FUNCTION FC 8 : VOID
TITLE = Ermittlung DB, DW, Laenge Anyzeiger
//Erstellung:
//Datum        Bearbeiter                                                 Version
//--------------------------------------------------------------------------------
//03.03.99     A.Geiger (gea)                                             01.00.00
//
//Änderungen:
//Nr. Datum    Bearb Beschreibung                                   Marke Version
//--------------------------------------------------------------------------------
//01  
//
//________________________________________________________________________________
//Funktion:
//
//Der Baustein ermittelt aus einem ANY-Zeiger:
//  Datenbausteinnummer
//  Datenwortnummer Beginn des Anyzeigers
//  Länge des Bereiches in Byte
//
AUTHOR : gea
FAMILY : AZO
VERSION : 0.0
VAR_INPUT
  in_Zeiger : ANY ;	//ANY-Zeiger
END_VAR
VAR_OUTPUT
  out_DB : INT ;	//Datenbausteinnummer
  out_DW : INT ;	//Anfangs-Datenwortnummer
  out_Laenge : INT ;	//Länge des Bereiches in Byte
END_VAR
BEGIN
NETWORK
TITLE = Ermittlung DB, DW, Laenge Anyzeiger
      L     P##in_Zeiger;
      LAR1;
      L     W [AR1,P#2.0];
      T     #out_Laenge;
      L     W [AR1,P#4.0];
      T     #out_DB;
      L     D [AR1,P#6.0];
      SRD   3;
      T     #out_DW;
END_FUNCTION

FUNCTION FC 10 : VOID
TITLE = Analogwert lesen/schreiben
//Erstellung:
//Datum        Bearbeiter                                                 Version
//--------------------------------------------------------------------------------
//06.08.97     G.Herkert (hkt)                                            01.00.00
//
//Änderungen:
//Nr. Datum    Bearb Beschreibung                                   Marke Version
//--------------------------------------------------------------------------------
//01  21.10.97 rh    Drahtbruchüberwachung ergänzt                        01.01.00
//02  05.12.97 rh    Adressen auf PEW und PAW geändert                    01.01.01
//03  25.11.98 gea   Simulation eingefügt                                 01.02.00
//04  29.03.99 gea   Fehlerbehebung Drahtbruchüberwachung                 01.02.01
//05  30.06.99 sra   Fehlerbehebung Drahtbruchüberwachung                 01.02.02
//06  19.02.00 sra   Unterscheidung Drahtbruchüberwachung                 01.02.03
//07  12.09.01 gea   Eingangsparameter in_E_A_Adresse als INT             01.03.00
//08  16.03.04 sra   nicht in Simulations-DB schreiben wenn Simul aus     01.03.01
//09  17.09.08 sra   Wago-System 750-466 erweitert                  (009) 01.04.00
//________________________________________________________________________________
//Funktion:
//
//Der Baustein liest den Wert eines Analogeinganges ein und normiert diesen. Die 
//Normierung erfolgt anhand der Vorgabe der Eingangsparameter Obergrenze und 
//Untergrenze.
//
//Hinweis:
//- bei Siemens-Baugruppen ist der Wert "MaxDigit" = 27648
//- bei Wago-Baugruppen 740-466 ist der Wert "MaxDigit" = 32760
//
//
AUTHOR : hkt
FAMILY : AZO
VERSION : 0.0
VAR_INPUT
  in_E_A : CHAR  := 'E';	//E = Eingang, A = Ausgang
  in_EA_Adresse : INT ;	//Ein-/Ausgangsadresse des Analogkanals
  in_OberGrenze : REAL ;	//Obergrenze des Ausgabewertes (z.B. Drucktransmitter: 2 bar)
  in_UnterGrenze : REAL ;	//Untergrenze des Ausgabewertes (z.B. Drucktransmitter: 0 bar)
  in_MaxDigit : REAL ;	//Digitwert den die Baugruppe bei der Obergrenze liefert z.B. 27648
  in_MinDigit : REAL ;	//Digitwert den die Baugruppe bei der Untergrenze liefert z.B. 0 bzw. -27648
  in_Typ : CHAR ;	//Z=Zentralbaugruppe, B=ET200B Analogmodul, W=Wago 750-466, sonstige
  in_Simulation : BOOL ;	//Simulation des Analogwertes über Eintrag in Datenbaustein
  in_DB_Simulation_EA : INT ;	//Simulation-DB des Analogwertes über Eintrag in Datenbaustein
END_VAR
VAR_IN_OUT
  io_Wert : REAL ;	//eingelesener und normierter Wert den die Baugrppe liefert
  io_Drahtbruch : BOOL ;	//Drahtbruchstoerung
END_VAR
VAR_TEMP
  MaxDigit_MinDigit : REAL ;
  E_MinDigit : REAL ;
  OG_UG : REAL ;
  Eingang_Real : REAL ;
  Pointer_EA_Adresse : DWORD ;
  Wert_analog : WORD ;
  DB_Sim : INT ;
END_VAR
BEGIN
NETWORK
TITLE = Zwischenwerte berechnen
      L     #in_MaxDigit;
      L     #in_MinDigit;
      -R;
      T     #MaxDigit_MinDigit;
      L     #in_OberGrenze;
      L     #in_UnterGrenze;
      -R;
      T     #OG_UG;
NETWORK
TITLE = Zeiger berechnen
// Zeiger auf EA-Adresse berechnen
      LAR1  P#0.0;
      L     #in_EA_Adresse;
      SLW   3;
      +AR1;
      LAR1;
      T     #Pointer_EA_Adresse;	//Zeiger auf EA-Adresse
      L     #in_DB_Simulation_EA;
      T     #DB_Sim;	//Zeiger auf EA-DB
NETWORK
TITLE = Analogwert einlesen
//Analogwert einlesen
//Formel:   Wert = UG + (OG-UG)*(E-MinDigit) / (MaxDigit-MminDigit)
      L     #in_E_A;
      L     'E';
      <>I;
      JC    NotE;
      A     #in_Simulation;
      JC    SIME;
      L     PIW [#Pointer_EA_Adresse];
      JU    WERE;	// (008)
SIME: OPN   DB [#DB_Sim];
      L     DBW [#Pointer_EA_Adresse];
WERE: T     #Wert_analog;
      A(;
      L     #in_Typ;	// Abfrage Drahtbruchüberwachung
      L     'Z';	// "Z" = Zentralbaugruppe
      ==I;
      );
      A(;
      L     #Wert_analog;	// 7FFF Ersatzwert für Drahtbruch
      L     W#16#7FFF;
      ==I;
      );
      O;
      A(;
      L     #in_Typ;	// Abfrage Drahtbruchüberwachung
      L     'B';	// "B" = ET200B Baugruppe
      ==I;
      );
      A(;
      L     #Wert_analog;	// 8000 Ersatzwert für Drahtbruch
      L     W#16#8000;
      ==I;
      );
      O;	// -> (009)
      A(;
      L     #in_Typ;	// Abfrage Kartentyp
      L     'W';	// "W" = Wago System 750-466
      ==I;	// Karte meldet mit den rechten 3 Bis ein Kurzschluss bzw. Überlauf
      );
      A(;
      L     #Wert_analog;
      L     W#16#7;
      AW;
      L     W#16#0;
      <>I;
      );	// <- (009)
      =     #io_Drahtbruch;
      L     #Wert_analog;
      ITD;
      DTR;
      T     #Eingang_Real;
      L     #Eingang_Real;
      L     #in_MinDigit;
      -R;
      T     #E_MinDigit;
      L     #OG_UG;
      L     #E_MinDigit;
      *R;
      L     #MaxDigit_MinDigit;
      /R;
      L     #in_UnterGrenze;
      +R;
      T     #io_Wert;
NotE: NOP   0;
NETWORK
TITLE = AnalogWert ausgeben:  
//AnalogWert ausgeben:
//Formel : A = MinDigit+(MaxDigit-MinDigit)*(Wert-UG)/ (Og-UG)
      L     #in_E_A;
      L     'A';
      <>I;
      JC    NotA;
      L     #io_Wert;
      L     #in_UnterGrenze;
      -R;
      L     #OG_UG;
      /R;
      L     #MaxDigit_MinDigit;
      *R;
      L     #in_MinDigit;
      +R;
      RND;
      T     #Wert_analog;
      A     #in_Simulation;
      JC    SIMA;
      T     PQW [#Pointer_EA_Adresse];
      JU    NotA;	// (008)
SIMA: OPN   DB [#DB_Sim];
      T     DBW [#Pointer_EA_Adresse];
NotA: NOP   0;
END_FUNCTION

FUNCTION FC 13 : VOID
TITLE = Baustein für Standardmerker
//Erstellung:
//Datum        Bearbeiter                                                 Version
//--------------------------------------------------------------------------------
//26.06.97     R.Schaffert (sra)                                          01.00.00
//
//Änderungen:
//Nr. Datum    Bearb Änderung                                       Marke  Version
//--------------------------------------------------------------------------------
//01  21.11.02 sra   Resetmerker eingefügt                          (001) 01.00.01
//02  30.08.12 pti   Lampe Steuerspannung ein eingefügt             (002) 01.01.00
//03  23.07.13 sra   Signale für Sicherung eingefügt                (003) 01.02.00
//04  05.12.13 sra   Signal Steuerspannung gelöscht                       01.03.00
//05  02.06.14 sra   M0.3 Reset ebenfalls gelöscht (zu Änderung 04)       01.03.01
//06  14.12.16 sra   Implement SFC51 to read battery information    (006) 01.04.00
//________________________________________________________________________________
//Funktion:
//  
//Der Baustein erzeugt folgende Standardsignale:
//- M 0.1 "konstant 1" Merker
//- M 0.2 "konstant 0" Merker
//- M 1.6 Melderentprelltakt (5 Sekunden) 
//- M 1.7 "Takt Timernachbildung" = in_Basistakt_Timer
//- MB4 Impulsmerker für Takte 2.0s, 1.6s, 1.0s, 0.8s, 0.5s, 0.4s, 0.2s, 0.1s
//  !!! MB 2 muss als Taktmerker in CPU parametriert werden  !!
//  Das MB 3 wird als Hilfsbyte zur Flankenauswertung benutzt
//- MW 6 Zeitwert Takt = in_Zeit_Basistakt_100ms
AUTHOR : sra
FAMILY : AZO
VERSION : 0.0
VAR_INPUT
  in_E_Sicherung_OK : BOOL ;	//Eingang Sicherung OK = Eingang Störung Sicherung
  in_Basistakt_Timer : BOOL ;	//Taktmerker für alle Zeitfunktionen (abhängig von Zykluszeit)
  in_Zeit_Basistakt_100ms : INT ;	//Zeitwert Basistakt in 100 ms
END_VAR
VAR_OUTPUT
  o_Lampe_Stoer_Sicherung : BOOL ;	//Ausgang der Lampe "Störung Sicherung"
  o_Stoerung_Sicherung : BOOL ;	//Störung Sicherung -> für Störbitzuweisung im DB34
END_VAR
VAR_TEMP
  NOP : INT ;
END_VAR
BEGIN
NETWORK
TITLE = Statische Merker  
      SET;
      S     M 0.1;
      R     M 0.2;
NETWORK
TITLE = Lampe "Störung Sicherung" und Störmeldung Sicherung
//(003)
      AN    #in_E_Sicherung_OK;
      =     #o_Lampe_Stoer_Sicherung;
      =     #o_Stoerung_Sicherung;
NETWORK
TITLE = Impulsmerker Takte
//Impulsmerker für Takte 2.0s, 1.6s, 1.0s, 0.8s, 0.5s, 0.4s, 0.2s, 0.1s
//positive Flankenauswertung auf die von der CPU erzeugten Takte
      L     MB 3;
      L     MB 2;
      T     MB 3;
      XOW;
      L     MB 2;
      AW;
      T     MB 4;
NETWORK
TITLE = Werte für Timernachbildung vorgeben
//!! Abhängig von Zykluszeit !! 
      A     #in_Basistakt_Timer;
      =     M 1.7;
      L     #in_Zeit_Basistakt_100ms;
      T     MW 6;
NETWORK
TITLE = Takt Melderentprellung
//Takt Melderentprellung
      AN    M 1.6;
      L     S5T#5S;
      SD    T 1;
      A     T 1;
      =     M 1.6;
NETWORK
TITLE = read Battery fault of CPU
//(006)
      CALL  SFC 51 (
           REQ                      := M 2.7,
           SZL_ID                   := W#16#392,
           INDEX                    := W#16#0,
           RET_VAL                  := DB3.DBW 62,
           BUSY                     := DB3.DBX 60.0,
           SZL_HEADER               := P#DB3.DBX 64.0,
           DR                       := P#DB3.DBX 68.0 BYTE 20);	// W#16#392 = Status of the backup batteries in a rack/module rack of a CPU after at least one battery has failed /  if ID = 392h -> Index is always 0
      L     DB3.DBB 68;
      L     0;
      <>I;
      =     DB3.DBX 31.3;
END_FUNCTION

FUNCTION FC 16 : VOID
TITLE = Sammelstoerung
//Erstellung:
//Datum        Bearbeiter                                                 Version
//--------------------------------------------------------------------------------
//26.07.99     M.Junker (jm)                                              01.00.00
//
//Änderungen:
//Nr. Datum    Bearb Änderung                                       Marke  Version
//--------------------------------------------------------------------------------
//01  14.09.99 jm    Spiegelung von PC ergänzt                            01.01.00
//02  06.10.99 jm    Störauswertung DWORD-weise                           01.02.00
//03  23.10.99 jm    QuitierungsDWORD von PC löschen                      01.03.00
//04  03.11.99 jm    Fehlerbeseitigung: QIP und DWORD                     01.03.01
//05  27.03.00 jm    Fehlerbeseitigung DWORD (Erstmeldung)                01.03.02
//06  19.04.05 jm    Fehlerbeseitigung Pointeradressen >8192(=>SLD) (006) 01.03.03
//07  23.02.06 jm    Quittierungs-DB Farbgrafik ist extern
//                   => Quittierung üder Kastor oder Farbgrafik     (007) 01.04.00
//08  23.03.06 sra   Einzelstörungsbereiche
//                   +Quitt.Erstwertmeldung über Quittierbereich         
//                   +Erstwertmeldung löschen ohne Störung          (008) 01.05.00
//09  10.05.06 sra   Fehlerbeseitigung zu Änderung 08               (009) 01.05.01
//10  11.05.06 sra   Änderung Quittierung von Farbgrafik            (010) 01.05.02
//11  05.10.06 jm    Anpassung für Siemens OP: extra Quittierbereich
//                   mit Flankenauswertung                          (011) 01.06.00
//12  01.04.08 jm    Steuerspannung entfernt, da Probleme mit OP-
//                   Quittierung (Problem: vorhandene Störung bei
//                   Steuerspannung aus am OP quittieren)           (012) 01.06.01
//13  16.11.15 sra   "Steuerspannung" in "Frg. Sammenstörung" geänd.(013) 01.06.02
//________________________________________________________________________________
//Beschreibung:
//
//!!!ACHTUNG: Parameter Anzahl Störungsbyte muß immer durch 4 teilbar sein!!!!
//
//Der Baustein überwacht einen definierbaren Teil eines Datenbaustein (DB34) in 
//dem alle Störmeldungen gesammelt werden. Sobald eine Störung vorhanden ist wird 
//das Signal "Sammelstörung" gebildet um damit z.B. eine Sammelstörlampe 
//anzusteuern. Der Parameter "Anzahl Störungsbyte" muß immer durch 4 teilbar sein
//
//In weiteren Bereichen weden die Datenblöcke "Erstmeldung", "Erstmeldung PC" und 
//Quittierung PC" mit der gleichen Größe wie der Störbereich benötigt.
//
//Funktion:
//Um bei der Störungsquittierung zur FG kompatibel zu sein werden die 
//Quittierungen, sobald die Störung verschwunden ist, von der SPS gelöscht.
//
//Die beiden Quittierungsbereiche (in DB34 für Kastor; in DB35 für SCADA) werden 
//mit ODER ausgewertet, d.h. die Störungen könnten von beiden Seiten quittiert 
//werden (wird normal nicht gemacht). Die Quittierbits werden hier so umkopiert, 
//daß sie immer in beiden Quittierungsbereichen auftauchen.
//=> es müssen immer beide Quittierbereiche angelegt sein
//=> an den Aggregat-Baustein werden die Bits aus dem DB35 angelegt
//
//OP:
//Siemens OPs müssen in einen extra Bereich quittieren, der hinter dem normalen 
//Standardbereichen im DB34 liegt. Im Anschluss folgt noch ein Bereich für die 
//Flankenauswertung. Bei positiver Flanke der Quittierung von OP wird die in den 
//Bereich der SCADA-Quittierung übertragen. In den OP Quittierbereich darf auf 
//gar keinen Fall die SPS schreiben. Wird kein OP verwendet so können die 
//OP-Bereiche aus dem DB34 weggelassen werden.
AUTHOR : jm
FAMILY : STANDARD
NAME : hsh
VERSION : 0.0
VAR_INPUT
  Conf_AckBySiemensOP : BOOL ;	//configuration bit: ackowledge done by Siemens OP (011)
  Stoerungstakt : BOOL ;	//Takt für Störauswertung
  Freigabe_Sammelstoerung : BOOL ;	//Freigabe Sammelstörung (ehemals Steuerspannung)
  Quittierung : BOOL ;	//Quittierung Fehlermeldung
  Stoerungs_DB : INT ;	//Stör-Datenbaustein
  Quittierungs_DB_SCADA : INT ;	//Quittier-Datenbaustein Farbgrafik
  Anzahl_Stoerungs_Byte : INT ;	//Anzahl Störungsbyte im Stör-Db (Blocklänge der 4 Bereiche)
  Offset_Stoerungs_Byte : INT ;	//Anfangs-DW der Störmeldungen im Stör-DB (wenn Bereich nicht bei Byte 0 anfängt)
  Adresse_Anfangswort : INT ;	//Adresse des ersten Datenwortes das ausgewertet wird
  Bereichslaenge : INT ;	//Länge des Bereiches der ausgewertet wird (!!Muss durch 4 teilbar sein!!)
END_VAR
VAR_IN_OUT
  Sammelstoerung : BOOL ;	//Sammelstörung
  Erstmeldung : BOOL ;	//Erstmeldung aktiv
  Erstmeldung_PC : BOOL ;	//Erstmeldung an PC
  Quittierung_PC : BOOL ;	//Quittierung von PC
END_VAR
VAR_TEMP
  Stoer_DB : INT ;	//Stoerungs-DB lokal
  Quit_DB : INT ;	//Quittierungs-DB extern
  Offsetende : INT ;	//= Störungsbyte + Offset
  SI : INT ;	//Störungsindex
  KI : INT ;	//Kopierindex
  SIP : INT ;	//Spiegelungsindex PC
  QIP : INT ;	//Quittierungsindex PC
  QIS : INT ;	//Quitierungsindex SCADA
  QIO : INT ;	//Quittierungsindex Siemens OP (011)
  KQIO : INT ;	//Kopie Quittierungsindex Siemens OP (011)
  StoerungsDWORD : DWORD ;	//Stoerungsdoppelwort
  KopieDWORD : DWORD ;	//Kopiedoppelwort
  SpiegelungsDWORD : DWORD ;	//Spiegelungsdoppelwort
  QuittierungsDWORD : DWORD ;	//Quittierungsdoppelwort
  QuitPC_DWORD : DWORD ;	//Quittierungsdoppelwort von PC
  QuitSCADA_DWORD : DWORD ;	//Quittierungsdoppelwort von SCADA
  QuitOP_DWORD : DWORD ;	//Quittierungdoppelwort von OP (011)
  KopieQuitOP_DWORD : DWORD ;	//Kopie Quittierungdoppelwort von OP (011)
  t_Erstmeldung_PC : BOOL ;	//Erstmeldung an PC
END_VAR
BEGIN
NETWORK
TITLE = Störauswertung aktiv?
//      ON    #Steuerspannung // (012)
//      SPB   FCEN                       // FunCtion ENd // (012)
      ON    #Stoerungstakt;
      JC    QUIT;	// QUITtierung Erstmeldung prüfen
NETWORK
TITLE = Variablen vorbelegen
//Minus 4 wegen DWORD-Auswertung
      CLR;
      =     #Sammelstoerung;
      =     #t_Erstmeldung_PC;
      L     #Offset_Stoerungs_Byte;
      L     #Adresse_Anfangswort;	// (008)
      +I;	// (008)
      L     #Bereichslaenge;	// (008)
      +I;
      T     #Offsetende;	//Offsetende = Offset + Anzahl // (007)
      L     #Offsetende;	// (007)
      L     4;
      -I;
      T     #SI;	//Stoerungsindex = Offsetende + Anzahl -4
      T     #QIS;	//Quittierungsindex SCADA = Stoerungsindex (007)
      L     #Offsetende;	// (007)
      L     #Anzahl_Stoerungs_Byte;	// (008)
      +I;
      L     4;
      -I;
      T     #KI;	//Kopierindex = Offsetende + Anzahl*2 -4
      L     #Offsetende;	// (007)
      L     #Anzahl_Stoerungs_Byte;
      +I;
      L     #Anzahl_Stoerungs_Byte;	// (008)
      +I;
      L     4;
      -I;
      T     #SIP;	//Spiegelungsindex PC = Offsetende + Anzahl*3 -4
      L     #Offsetende;	// (007)
      L     #Anzahl_Stoerungs_Byte;
      +I;
      L     #Anzahl_Stoerungs_Byte;
      +I;
      L     #Anzahl_Stoerungs_Byte;	// (008)
      +I;
      L     4;
      -I;
      T     #QIP;	//Quittierungsindex PC = Offsetende + Anzahl*4 -4
// >>>>>>>>>> (011)
      L     #Offsetende;
      L     #Anzahl_Stoerungs_Byte;
      +I;
      L     #Anzahl_Stoerungs_Byte;
      +I;
      L     #Anzahl_Stoerungs_Byte;
      +I;
      L     #Anzahl_Stoerungs_Byte;
      +I;
      L     4;
      -I;
      T     #QIO;	//Quittierungsindex OP = Offsetende + Anzahl*5 -4
      L     #Offsetende;
      L     #Anzahl_Stoerungs_Byte;
      +I;
      L     #Anzahl_Stoerungs_Byte;
      +I;
      L     #Anzahl_Stoerungs_Byte;
      +I;
      L     #Anzahl_Stoerungs_Byte;
      +I;
      L     #Anzahl_Stoerungs_Byte;
      +I;
      L     4;
      -I;
      T     #KQIO;	//Kopie Quittierungsindex OP = Offsetende + Anzahl*6 -4
// <<<<<<<<<< (011)
NETWORK
TITLE = Störungs-/Kopie-/Spiegelungs-/QuittierungsDWORD(OP) laden
      L     #Stoerungs_DB;
      T     #Stoer_DB;
      L     #Quittierungs_DB_SCADA;	// (007)
      T     #Quit_DB;	// (007)
SLOP: OPN   DB [#Stoer_DB];
      L     #SI;
      SLD   3;	// (006)
      LAR1;
      L     DBD [AR1,P#0.0];
      T     #StoerungsDWORD;
      L     #KI;
      SLD   3;	// (006)
      LAR1;
      L     DBD [AR1,P#0.0];
      T     #KopieDWORD;
      L     #SIP;
      SLD   3;	// (006)
      LAR1;
      L     DBD [AR1,P#0.0];
      T     #SpiegelungsDWORD;
      L     #QIP;
      SLD   3;	// (006)
      LAR1;
      L     DBD [AR1,P#0.0];
      T     #QuitPC_DWORD;	// (007)
///*(007)
      L     L#0;	// (011)
      T     #QuitSCADA_DWORD;
      L     #Quittierungs_DB_SCADA;	// (011)
      L     0;
      ==I;	// (011)
      JC    KQ1;	// (011) kein Quittierungsbaustein vorhanden
      OPN   DB [#Quit_DB];
      L     #QIS;
      SLD   3;
      LAR1;
      L     DBD [AR1,P#0.0];
      T     #QuitSCADA_DWORD;
      OPN   DB [#Stoer_DB];
//(007)*/
// >>>>>>>>>> (011)
      L     0;
      T     #QuitOP_DWORD;	// vorbelegen, falls nicht vorhanden
      AN    #Conf_AckBySiemensOP;
      JC    NOPA;	// No OP Acknowledge
      L     #QIO;
      SLD   3;
      LAR1;
      L     DBD [AR1,P#0.0];
      T     #QuitOP_DWORD;
      L     #KQIO;
      SLD   3;
      LAR1;
      L     DBD [AR1,P#0.0];
      T     #KopieQuitOP_DWORD;
NOPA: NOP   0;	// No OP Acknowledge
// <<<<<<<<<< (011)
KQ1:  NOP   0;
NETWORK
TITLE = Pos.Flanke Quittierung OP
//(011)
      AN    #Conf_AckBySiemensOP;
      JC    NPOA;	// No Processing of Op Acknowledge
      L     #QuitOP_DWORD;	// -
      L     #KopieQuitOP_DWORD;	// |
      XOD;	// | positive Flanke Quittierung OP
      L     #QuitOP_DWORD;	// |
      AD;	// -
      L     #QuitSCADA_DWORD;
      OD;
      T     #QuitSCADA_DWORD;	// => Quittierung in QuitSCADA setzen
      L     #QuitOP_DWORD;
      T     #KopieQuitOP_DWORD;	// => Hilfsmerker Flanke (Kopie ALT)
NETWORK
TITLE = Quittierung OP DWORD nach Kopiebyte
//(011)
      L     #KQIO;
      SLD   3;
      LAR1;
      L     #KopieQuitOP_DWORD;
      T     DBD [AR1,P#0.0];	// => Quittierung OP merken
NPOA: NOP   0;
NETWORK
TITLE = Sammelstörung
      L     #StoerungsDWORD;
      L     0;
      <>D;
      A     #Freigabe_Sammelstoerung;	// (012)
      S     #Sammelstoerung;
NETWORK
TITLE = Erstwertmeldung
      L     #StoerungsDWORD;
      L     #KopieDWORD;
      XOD;
      L     #StoerungsDWORD;
      AD;
      L     0;
      <>D;
      A     #Freigabe_Sammelstoerung;	// (012)
      S     #Erstmeldung;
NETWORK
TITLE = Erstwertmeldung an PC
      L     #StoerungsDWORD;
      L     #SpiegelungsDWORD;
      <>D;
      S     #t_Erstmeldung_PC;
NETWORK
TITLE = StoerungsDWORD nach Kopiebyte
      L     #KI;
      SLD   3;	// (006)
      LAR1;
      L     #StoerungsDWORD;
      T     DBD [AR1,P#0.0];
NETWORK
TITLE = neue Quittierung?
//(008)
      L     #QuitSCADA_DWORD;
      L     #QuitPC_DWORD;
      XOD;
      L     0;
      <>D;
      R     #Erstmeldung;
NETWORK
TITLE = QuittierungsDWORD bilden
//(007)
      L     #QuitPC_DWORD;	// (010)
      L     #SpiegelungsDWORD;	// (010)
      AD;	// (010)
      L     #QuitSCADA_DWORD;
      OD;
      T     #QuittierungsDWORD;	// Quittierung von Kastor oder SCADA
NETWORK
TITLE = QuittierungsDWORD löschen
      L     #StoerungsDWORD;
      L     #QuittierungsDWORD;
      AD;
      T     #QuittierungsDWORD;
NETWORK
TITLE = QuittierungsDWORD PC und SCADA löschen
      L     #QIP;
      SLD   3;	// (006)
      LAR1;
      L     #QuittierungsDWORD;
      T     DBD [AR1,P#0.0];	// PC Quittierung
      L     #Quittierungs_DB_SCADA;	// (011)
      L     0;	// (011)
      ==I;	// (011)
      JC    KQ2;	// (011) kein Quittierungsbaustein vorhanden
///*(007)
      OPN   DB [#Quit_DB];
      L     #QIS;
      SLD   3;
      LAR1;
      L     #QuittierungsDWORD;
      T     DBD [AR1,P#0.0];	// SCADA Quittierung
//(007)*/
KQ2:  NOP   0;
NETWORK
TITLE = Störungsschleife von (Anzahl - 4) bis 0
//Minus 4 wegen DWORD-Auswertung
// >>>>>>>>>> (011)
      L     #KQIO;
      L     4;
      -I;
      T     #KQIO;
      L     #QIO;
      L     4;
      -I;
      T     #QIO;
// <<<<<<<<<< (011)
///*(007)
      L     #QIS;
      L     4;
      -I;
      T     #QIS;
//(007)*/
      L     #QIP;
      L     4;
      -I;
      T     #QIP;
      L     #SIP;
      L     4;
      -I;
      T     #SIP;
      L     #KI;
      L     4;
      -I;
      T     #KI;
      L     #SI;
      L     4;
      -I;
      T     #SI;
      L     #Offset_Stoerungs_Byte;
      L     #Adresse_Anfangswort;	// (008)
      +I;	// (008)
      L     #SI;	// (008)
      <=I;	// (008) (009)
      JC    SLOP;	// Störungs LOOP
NETWORK
TITLE = Störauswertung für PC aktiv?
      O     #Erstmeldung_PC;
      O     #Quittierung_PC;
      JC    QUIT;	//QUITtierung
      A     #t_Erstmeldung_PC;
      S     #Erstmeldung_PC;
NETWORK
TITLE = Erstmeldung quittiert?
QUIT: A     #Quittierung;	//QUITtierung
      ON    #Sammelstoerung;	// (008)
      R     #Erstmeldung;
      A     #Quittierung_PC;
      R     #Erstmeldung_PC;
      NOP   0;
END_FUNCTION

FUNCTION FC 20 : VOID
TITLE = Block for motor actuation and fault monitoring
//Erstellung:
//Datum        Bearbeiter                                                 Version
//--------------------------------------------------------------------------------
//26.06.97     H.Rüttling (rh)                                            01.00.00
//
//Änderungen:
//Nr. Datum    Bearb Änderung                                       Marke  Version
//--------------------------------------------------------------------------------
//01  09.02.99 sra   Einfügen der Handbedienuung                    ()    01.01.00
//02  16.04.99 sra   Fehlerbeseitigung Störungsquittierung          ()    01.01.01
//03  23.07.99 sra   Ausg. wird auch bei Simulation gesetzt         ()    01.01.02
//04  19.10.99 sra   "in" Reparaturschalter gelöscht                ()    01.02.00
//05  03.11.99 hus   Parameter eingefügt "FU in Betrieb"            ()    01.03.00
//06  18.09.00 sra   komplette Überarbeitung / neue Struktur        ()    02.00.00
//07  08.11.02 sra   Änderung Betriebsstundenzähler (zählt falsch)  (007) 02.01.00
//08  31.10.05 sra   Ansteuerung Handbedienung im Automode rücksetz.
//                   Handbedienung zentral sperren                  (008) 02.02.00
//09  04.09.06 sra   Änderung Störungsquittierung                   (009) 02.03.00
//10  20.11.07 gea   Handmode zurücksetzen wenn Handmode gesperrt   (010) 02.03.01
//11  18.02.09 kmj   Objektststatus für OP ergänzt                  (011) 02.04.00
//12  20.03.09 kal   Objektststatus für OP ergänzt (überarbeitet)   (012) 02.04.01
//13  05.12.13 sra   "Anlage ein" eingefügt (Not-Aus-Konzept)       (013) 02.05.00
//________________________________________________________________________________
//Funktion:
//
//-Der Baustein steuert den Ablauf eines Motors mit 1 Ausgang und 1 Eingang durch 
// setzten des Eingangsparameters "in_Ansteuerung_Motor".
//
//-Der Ausgang wird nur angesteuert wenn der Eingang "in_Anlage_ein" = true
// ist. Diese Funktion ist vorhanden, um bei einem Not-Halt die Anlage vor 
// unkontrolliertem Einschalten zu schützen. 
//
//-Ist in der Motorstruktur die Taktfunktion freigegeben wird bei Freigabe des 
// Motors der Ausgang entsprechend der Impuls-/Pausezeit angesteuert.
// !!Der Baustein arbeitet nur mit vollen Sekunden!!
//
//-Der Baustein überwacht den Zustand des Ausgangs und des Eingangs und generiert 
// nach Ablauf der "Sollzeit Störung" eine Störmeldung
//
//-Ist das Bit "Simulation" auf TRUE, so wird der Eingang simuliert.
//
//-Ist die Kennung "Betriebsstundenzähler_ein" aktiviert werden die Laufzeit 
// des Motors aufsummiert. Dies erfolgt mit setzen des Ausgangs.
//
//-Der Baustein kopiert die Parameter "in_Eingang_Motor", "io_Ausgang_Motor", 
// "in_Quitt_Stoerung" und "io_Stoerung" in die angegebene Datenstruktur zur 
// Visualisierung auf einem Farbgrafiksystem. Diese Parameter müssen folglich 
// nicht mehr extern umkopiert werden.
//
//-Ist der Parameter "in_Handbedienung_erlaubt" angewählt kann der Motor über 
// eine Farbgrafik oder ein Bedienterminal manuell angesteuert werden
//
AUTHOR : rh
FAMILY : AZO
VERSION : 0.0
VAR_INPUT
  in_Handbedienung_erlaubt : BOOL ;	//1 = manual operation permitted, 0 = manual operation not permitted/locked
  in_Quitt_Stoerung_noetig : BOOL ;	//1 = fault acknowledgement required, 0 = automatic fault acknowledgement
  in_Anlage_ein : BOOL ;	//Anlage bzw. Anlagenbereich nach Not-Halt freigegeben
  in_Quitt_Stoerung : BOOL ;	//Fault acknowledgement when fault_acknowledgement_required = 1
  in_Ansteuerung_Motor : BOOL ;	//Actuation of motor in automatic mode
  in_Eingang_Motor : BOOL ;	//Input of motor
END_VAR
VAR_IN_OUT
  io_Ausgang_Motor : BOOL ;	//Output of motor
  io_Motor_in_Betrieb : BOOL ;	//Signal "motor in operation"
  io_Stoerung : BOOL ;	//Signal "motor fault"
  io_Motorstruktur : ANY ;	//ANY pointer of motor structure
END_VAR
VAR_TEMP
  Freigabe_Takt : BOOL ;
  Start_mit_Impuls : BOOL ;
  Dauertakt : BOOL ;
  Taktausgang : BOOL ;
  Taktanzahl_erreicht : BOOL ;
  Diskrepanz : BOOL ;
  Impulszeit : REAL ;
  Pausezeit : REAL ;
  Sollanzahl_Takte : INT ;
  Zeitzaehler : REAL ;
  Taktzaehler : INT ;
  Objektstatus : INT ;
END_VAR
BEGIN
NETWORK
TITLE = Anfangs-DW der Struktur aus ANY-Zeiger auslesen
      L     P##io_Motorstruktur;
      LAR2;
      L     D [AR2,P#6.0];
      LAR2;
NETWORK
TITLE = Simulation
      AN    DIX [AR2,P#3.5];	// Simulation ein (Struktur)
      JC    ESIM;
      A     #io_Ausgang_Motor;
      =     #in_Eingang_Motor;
ESIM: NOP   0;
NETWORK
TITLE = Umschaltung Hand-/Automatikmode 
      A     DIX [AR2,P#2.7];	// Handmode von Farbgrafik (Struktur)
      AN    DIX [AR2,P#3.1];	// Handmode gesperrt (Struktur)
      AN    M 0.0;	// Handbedienung zentral sperren (008)
      S     DIX [AR2,P#2.6];	// Handmode zu Farbgrafik (Struktur)
      ON    DIX [AR2,P#2.7];	// Handmode von Farbgrafik (Struktur)
      ON    #in_Handbedienung_erlaubt;
      O     M 0.0;	// Handbedienung zentral sperren (008)
      O     DIX [AR2,P#3.1];	// Handmode gesperrt (Struktur)//(010)
      R     DIX [AR2,P#2.6];	// Handmode zu Farbgrafik (Struktur)
      R     DIX [AR2,P#2.7];	// Handmode zu Farbgrafik (Struktur) (008)
NETWORK
TITLE = Ansteuerung Handmode zurücksetzen
//(008) 
      AN    DIX [AR2,P#2.6];	// Handmode zu Farbgrafik (Struktur)
      R     DIX [AR2,P#3.0];	// Ansteuerung Handmode von Farbgrafik (Struktur)
NETWORK
TITLE = Daten für Takt in temporäre Variablen laden
      A     #in_Anlage_ein;	// (013)
      A     #in_Ansteuerung_Motor;
      A     DIX [AR2,P#3.6];	// Freigabe Takt (Struktur)
      =     #Freigabe_Takt;
      A     DIX [AR2,P#3.2];	// Start mit Impuls (Struktur)
      =     #Start_mit_Impuls;
      A     DIX [AR2,P#3.3];	// Taktanzahl erreicht (Struktur)
      =     #Taktanzahl_erreicht;
      A     DIX [AR2,P#3.4];	// Dauertakt (Struktur)
      =     #Dauertakt;
      A     DIX [AR2,P#3.7];	// Taktausgang (Struktur)
      =     #Taktausgang;
      L     DID [AR2,P#8.0];	// Impulszeit (Struktur)
      T     #Impulszeit;
      L     DID [AR2,P#12.0];	// Pausezeit (Struktur)
      T     #Pausezeit;
      L     DIW [AR2,P#20.0];	// Sollanzahl Takte (Struktur)
      T     #Sollanzahl_Takte;
      L     DID [AR2,P#16.0];	// Impuls-/Pausezähler (Struktur)
      T     #Zeitzaehler;
      L     DIW [AR2,P#22.0];	// Taktzähler (Struktur)
      T     #Taktzaehler;
NETWORK
TITLE = Takt generieren
      CALL  FC 2 (
           in_Freigabe              := #Freigabe_Takt,
           in_Rueckmeldung          := #in_Eingang_Motor,
           in_Start_mit_Impuls      := #Start_mit_Impuls,
           in_Dauertakt             := #Dauertakt,
           in_Impuls                := M 4.5,
           in_Impulszeit_in_100ms   := 10,
           in_Impulszeit            := #Impulszeit,
           in_Pausezeit             := #Pausezeit,
           in_Sollanzahl_Takte      := #Sollanzahl_Takte,
           io_Taktausgang           := #Taktausgang,
           io_Taktanzahl_erreicht   := #Taktanzahl_erreicht,
           io_Zeitzaehler           := #Zeitzaehler,
           io_Taktzaehler           := #Taktzaehler);
NETWORK
TITLE = Ansteuerung Ausgang des Motors
      A     #in_Anlage_ein;	// (013)
      AN    DIX [AR2,P#2.2];	// Motor gesperrt (Struktur)
      A(;
      AN    #in_Quitt_Stoerung_noetig;
      O;
      A     #in_Quitt_Stoerung_noetig;	// Wenn die Stoerung quittiert werden muß 
      AN    #io_Stoerung;	// wird der Ausgang bei einer anstehenden
      );	// Stoerung zurück gesetzt
      A(;
      AN    DIX [AR2,P#2.6];	// Automatikmode zu Farbgrafik (Struktur)
      AN    DIX [AR2,P#3.6];	// Freigabe Takt (Struktur)
      A     #in_Ansteuerung_Motor;
      O;
      AN    DIX [AR2,P#2.6];	// Automatikmode zu Farbgrafik (Struktur)
      A     DIX [AR2,P#3.6];	// Freigabe Takt (Struktur)
      A     #Taktausgang;
      O;
      A     DIX [AR2,P#2.6];	// Handmode zu Farbgrafik (Struktur)
      A     DIX [AR2,P#3.0];	// Ansteuerung Handmode von Farbgrafik (Struktur)
      );
      O;
      A     #in_Anlage_ein;	// (013)
      A     DIX [AR2,P#24.0];	// FU in Betrieb (Struktur)              
      A     #io_Ausgang_Motor;	// Ausschalten nur möglich, wenn Bit = 0 
      =     #io_Ausgang_Motor;
NETWORK
TITLE = Betriebsmeldung
      A     #io_Ausgang_Motor;
      A     #in_Eingang_Motor;
      =     #io_Motor_in_Betrieb;
NETWORK
TITLE = Diskrepanz feststellen
      A     #io_Ausgang_Motor;
      AN    #in_Eingang_Motor;
      O;
      A     #in_Eingang_Motor;
      AN    #io_Ausgang_Motor;
      =     #Diskrepanz;
NETWORK
TITLE = Störungszähler
      A     #in_Quitt_Stoerung_noetig;
      AN    #in_Quitt_Stoerung;
      A     #io_Stoerung;
      O;
      A     #Diskrepanz;
      AN    #in_Quitt_Stoerung;	// (009)
      O;	// (009)
      AN    #in_Quitt_Stoerung_noetig;	// (009)
      A     #Diskrepanz;	// (009)
      JC    SZ1;
      L     0;	// Wenn keine Diskrepanz dann Zähler löschen
      T     DIW [AR2,P#6.0];	// Istzeit Störung (Struktur)
      JU    ESZ;
// Störungszähler in jeder Sekunde erhöhen
SZ1:  O     #io_Stoerung;
      ON    M 4.5;	// Sekundenimpuls (Standardmerker)
      JC    ESZ;
      L     DIW [AR2,P#6.0];	// Istzeit Störung (Struktur)
      INC   1;
      T     DIW [AR2,P#6.0];	// Istzeit Störung (Struktur)
ESZ:  NOP   0;
NETWORK
TITLE = Störmeldung ausgeben
      L     DIW [AR2,P#6.0];	// Istzeit Störung (Struktur)
      L     DIW [AR2,P#4.0];	// Sollzeit Störung (Struktur)
      >=I;
      =     #io_Stoerung;
NETWORK
TITLE = Stoerung quittieren
      O     #Diskrepanz;	// Stoerung steht noch an
      ON    #io_Stoerung;
      JC    ESQ;
      ON    #in_Quitt_Stoerung_noetig;	// Stoerung muß quittiert werden ?
      JC    SQ1;	// Stoerung muß nicht quittiert werden
      A     #in_Quitt_Stoerung;
SQ1:  R     #io_Stoerung;
ESQ:  NOP   0;
NETWORK
TITLE = Betriebsstundenzähler
//jede Sekunde wird der Sekundenzähler erhöht und beim erreichen von 3600 
//Sekunden wird eine Betriebsstunde addiert. (nur über Gleitpunktwert zu ungenau)
      ON    DIX [AR2,P#0.3];	// Kennung Betriebsstundenzähler ein (Struktur)
      ON    #io_Ausgang_Motor;
      ON    M 4.5;	// Sekundentakt
      JC    EBSZ;
      L     DIW [AR2,P#44.0];	// Betriebsstunden Sekundenzähler bis 3600 (007)
      L     1;	// (007)
      +I;	// (007)
      T     DIW [AR2,P#44.0];	// Betriebsstunden Sekundenzähler bis 3600 (007)
      L     3600;	// (007)
      <I;	// (007)
      JC    EBSZ;	// (007)
      L     DID [AR2,P#32.0];	// Betriebsstundenzähler (007)
      L     1.000000e+00;	// (007)
      +R;	// (007)
      T     DID [AR2,P#32.0];	// Betriebsstundenzähler (007)
      L     0;	// (007)
      T     DIW [AR2,P#44.0];	// Betriebsstunden Sekundenzähler bis 3600 (007)
EBSZ: NOP   0;
NETWORK
TITLE = Betriebsstundenzähler zurücksetzten
      AN    DIX [AR2,P#30.0];	// Reset Betriebsstundenzähler (Struktur)
      JC    E_RB;
      L     0.000000e+00;
      T     DID [AR2,P#32.0];	// Betriebsstundenzähler (Struktur)
      CLR;
      =     DIX [AR2,P#30.0];	// Reset Betriebsstundenzähler (Struktur)
E_RB: NOP   0;
NETWORK
TITLE = Warnmeldung Betriebsstundenzähler erzeugen
      A(;
      L     DID [AR2,P#32.0];	// Betriebsstundenzähler (Struktur)
      L     DID [AR2,P#36.0];	// Sollzeit Warnung (Struktur)
      >R;
      );
      A(;
      L     DID [AR2,P#36.0];	// Sollzeit Warnung (Struktur)
      L     0.000000e+00;
      <>R;
      );
      =     DIX [AR2,P#30.1];	// Warnmeldung Betriebsstundenzähler (Struktur)
NETWORK
TITLE = Alarmmeldung Betriebsstundenzähler erzeugen
      A(;
      L     DID [AR2,P#32.0];	// Betriebsstundenzähler (Struktur)
      L     DID [AR2,P#40.0];	// Sollzeit Alarm (Struktur)
      >R;
      );
      A(;
      L     DID [AR2,P#40.0];	// Sollzeit Alarm (Struktur)
      L     0.000000e+00;
      <>R;
      );
      =     DIX [AR2,P#30.2];	// Warnmeldung Betriebsstundenzähler (Struktur)
NETWORK
TITLE = Objektstatus für Visualisation OP // (011)(012)
//Stati:
//-------
//1 = nicht in Betrieb, keine Störung ==> Farborschlag weiß
//5 = angesteuert, in Betrieb, keine Störung ==> Farbvorschalg grün
//9 = angesteuert, nicht in Betrieb, keine Störung ==> Farbvorschalg grau
//16 = Störung ==> Farbvorschalg rot
// 1 = nicht in Betrieb, keine Störung ==> Farborschlag weiß
      L     1;
      AN    #io_Ausgang_Motor;
      AN    #in_Eingang_Motor;
      AN    #io_Stoerung;
      JC    disp;
// 5 = angesteuert, in Betrieb, keine Störung ==> Farbvorschalg grün
      L     5;
      A     #io_Ausgang_Motor;
      A     #in_Eingang_Motor;
      AN    #io_Stoerung;
      JC    disp;
// 9 = angesteuert, nicht in Betrieb, keine Störung ==> Farbvorschalg grau
      L     9;
      A     #io_Ausgang_Motor;
      AN    #in_Eingang_Motor;
      AN    #io_Stoerung;
      JC    disp;
// 16 = Störung ==> Farbvorschalg rot
      L     16;
      A     #io_Stoerung;
      JC    disp;
      L     0;
disp: T     #Objektstatus;
NETWORK
TITLE = Daten in Struktur speichern
      A     #in_Anlage_ein;	// (013)
      =     DIX [AR2,P#46.0];	// (013) Anlage ein (Struktur)
      A     #in_Eingang_Motor;
      =     DIX [AR2,P#2.1];	// Eingang Motor (Struktur)
      A     #io_Ausgang_Motor;
      =     DIX [AR2,P#2.0];	// Ausgang Motor (Struktur)
      A     #io_Motor_in_Betrieb;
      =     DIX [AR2,P#2.4];	// Motor in Betrieb (Struktur)
      A     #io_Stoerung;
      =     DIX [AR2,P#2.5];	// Störung (Struktur)
      A     #Taktanzahl_erreicht;
      =     DIX [AR2,P#3.3];	// Taktanzahl erreicht (Struktur)
      A     #Taktausgang;
      =     DIX [AR2,P#3.7];	// Taktausgang (Struktur)
      L     #Zeitzaehler;
      T     DID [AR2,P#16.0];	// Impuls-/Pausezähler (Struktur)
      L     #Taktzaehler;
      T     DIW [AR2,P#22.0];	// Taktzähler (Struktur)
      L     #Objektstatus;	// (011)
      T     DIW [AR2,P#48.0];	// #Objektstatus  (Struktur)   // (011)
NETWORK
TITLE = ENDE
      NOP   0;
END_FUNCTION

FUNCTION FC 21 : VOID
TITLE = Block for valve actuation and fault monitoring
//Erstellung:
//Datum        Bearbeiter                                                 Version
//--------------------------------------------------------------------------------
//26.06.97     H.Rüttling (rh)                                            01.00.00
//
//Änderungen:
//Nr. Datum    Bearb Änderung                                       Marke  Version
//--------------------------------------------------------------------------------
//01  09.02.99 sra   Einfügen der Handbedienuung                    ()    01.01.00
//02  16.04.99 sra   Fehlerbeseitigung Störungsquittierung          ()    01.01.01
//03  21.05.99 jm    Ventiltyp 0 eingefügt                          ()    01.02.00
//04  23.07.99 sra   Ausg. wird auch bei Simulation gesetzt         ()    01.02.01
//06  18.09.00 sra   komplette Überarbeitung / neue Struktur        ()    02.00.00
//07  31.10.05 sra   Ansteuerung Handbedienung im Automode rücksetz.
//                   Handbedienung zentral sperren                  (007) 02.01.00
//08  04.09.06 sra   Änderung Störungsquittierung                   (008) 02.02.00
//09  18.02.09 kmj   Objektststatus für OP ergänzt                  (009) 02.03.00
//10  20.03.09 kal   Objektststatus für OP ergänzt (überarbeitet)   (010) 02.03.01
//11  25.03.09 kal   1A0E-Objekt kann verzögert "in Betrieb" melden (011) 02.03.02
//12  25.03.09 kal   INC nach + geändert                            (012) 02.03.03
//13  20.11.07 gea   Handmode zurücksetzen wenn Handmode gesperrt   (013) 02.03.04
//14  14.07.09 kal   Objektstatus überarbeitet                      (014) 02.03.05
//15  05.12.13 sra   "Anlage ein" eingefügt (Not-Aus-Konzept)       (015) 02.04.00
//________________________________________________________________________________
//Funktion:
//
//-Der Parameter VENTIL_TYP unterscheidet zwischen 4 verschiedenen Ventiltypen
// Typ 0 = Ventil ohne Rückmeldung
// Typ 1 = Ventil oder Klappe mit der Rückmeldung angesteuert und nicht 
//        angesteuert: 1. Ausgang auf, Eingang auf, Eingang zu
//                     2. Ausgang zu , Eingang zu , Eingang auf
// TYP 2 = Ventil oder Klappe mit der Rückmeldung angesteuert
//                     1. Ausgang auf, Eingang auf
//                     2. Ausgang zu , Eingang zu 
// TYP 3 = Ventil oder Klappe mit der Rückmeldung nicht angesteuert
//                     1. Ausgang auf, Eingang zu
//                     2. Ausgang zu , Eingang auf 
//
//-Der Baustein steuert den Ablauf eines Ventils mit 1 Ausgang und 0-2 Eingängen
// durch setzten des Eingangsparameters "in_Ansteuerung_Ventil".
//
//-Der Ausgang wird nur angesteuert wenn der Eingang "in_Anlage_ein" = true
// ist. Diese Funktion ist vorhanden, um bei einem Not-Halt die Anlage vor 
// unkontrolliertem Einschalten zu schützen. 
//
//-Ist in der Ventilstruktur die Taktfunktion freigegeben wird bei Freigabe des 
// Ventils der Ausgang entsprechend der Impuls-/Pausezeit angesteuert.
//
//-Der Baustein überwacht den Zustand des Ausgangs und der Eingänge und generiert 
// nach Ablauf der "Sollzeit Störung" eine Störmeldung
//
//-Ist das Bit "Simulation" auf TRUE, so werden die Eingänge simuliert.
//
//-Ist die Kennung "Schalthäufigkeitszähler_ein" aktiviert werden die
// Ansteuerungen des Ventils aufsummiert. Dies erfolgt mit setzen des Ausgangs.
//
//-Der Baustein kopiert die Parameter "in_Eingang_...", "io_Ausgang_Ventil", 
// "in_Quitt_Stoerung" und "io_Stoerung" in die angegebene Datenstruktur zur 
// Visualisierung auf einem Farbgrafiksystem. Diese Parameter müssen folglich 
// nicht mehr extern umkopiert werden.
//
//-Ist der Parameter "in_Handbedienung_erlaubt" angewählt kann das Ventil über 
// eine Farbgrafik oder ein Bedienterminal manuell angesteuert werden
//
AUTHOR : rh
FAMILY : AZO
VERSION : 0.0
VAR_INPUT
  in_Ventil_Typ : INT ;	//see Functional description below
  in_Handbedienung_erlaubt : BOOL ;	//1 = manual operation permitted, 0 = manual operation not permitted/locked
  in_Quitt_Stoerung_noetig : BOOL ;	//1 = fault acknowledgement required, 0 = automatic fault acknowledgement
  in_Quitt_Stoerung : BOOL ;	//Fault acknowledgement when fault_acknowledgement_required = 1
  in_Anlage_ein : BOOL ;	//Anlage bzw. Anlagenbereich nach Not-Halt freigegeben
  in_Ansteuerung_Ventil : BOOL ;	//Actuation of valve in automatic mode
  in_Eingang_angesteuert : BOOL ;	//Valve intake when actuated
  in_Eingang_nicht_angest : BOOL ;	//Valve intake when not actuated
END_VAR
VAR_IN_OUT
  io_Ausgang_Ventil : BOOL ;	//Valve outlet
  io_Ventil_in_Betrieb : BOOL ;	//Signal "valve in operation" (actuated)
  io_Stoerung : BOOL ;	//Signal "valve fault"
  io_Ventilstruktur : ANY ;	//ANY pointer of valve structure
END_VAR
VAR_TEMP
  Freigabe_Takt : BOOL ;
  Rueckmeldung : BOOL ;
  Start_mit_Impuls : BOOL ;
  Dauertakt : BOOL ;
  Taktausgang : BOOL ;
  Taktanzahl_erreicht : BOOL ;
  Diskrepanz : BOOL ;
  positive_Flanke : BOOL ;
  Impulszeit : REAL ;
  Pausezeit : REAL ;
  Sollanzahl_Takte : INT ;
  Zeitzaehler : REAL ;
  Taktzaehler : INT ;
  Objektstatus : INT ;
END_VAR
BEGIN
NETWORK
TITLE = Anfangs-DW der Struktur aus ANY-Zeiger auslesen
      L     P##io_Ventilstruktur;
      LAR2;
      L     D [AR2,P#6.0];
      LAR2;
NETWORK
TITLE = Simulation
      AN    DIX [AR2,P#3.5];	// Simulation ein (Struktur)
      JC    ESIM;
      A     #io_Ausgang_Ventil;
      =     #in_Eingang_angesteuert;
      AN    #io_Ausgang_Ventil;
      =     #in_Eingang_nicht_angest;
      L     #in_Ventil_Typ;
      L     3;
      <>I;
      JC    ESIM;
      CLR;
      =     #in_Eingang_angesteuert;
      AN    #io_Ausgang_Ventil;
      =     #in_Eingang_nicht_angest;
ESIM: NOP   0;
NETWORK
TITLE = Umschaltung Hand-/Automatikmode 
      A     DIX [AR2,P#2.7];	// Handmode von Farbgrafik (Struktur)
      AN    DIX [AR2,P#3.1];	// Handmode gesperrt (Struktur)
      AN    M 0.0;	// Handbedienung zentral sperren (007)
      S     DIX [AR2,P#2.6];	// Handmode zu Farbgrafik (Struktur)
      ON    DIX [AR2,P#2.7];	// Handmode von Farbgrafik (Struktur)
      ON    #in_Handbedienung_erlaubt;
      O     M 0.0;	// Handbedienung zentral sperren (007)
      O     DIX [AR2,P#3.1];	// Handmode gesperrt (Struktur)//(013)
      R     DIX [AR2,P#2.6];	// Handmode zu Farbgrafik (Struktur)
      R     DIX [AR2,P#2.7];	// Handmode von Farbgrafik (Struktur) (007)
NETWORK
TITLE = Ansteuerung Handmode zurücksetzen
//(007) 
      AN    DIX [AR2,P#2.6];	// Handmode zu Farbgrafik (Struktur)
      R     DIX [AR2,P#3.0];	// Ansteuerung Handmode von Farbgrafik (Struktur)
NETWORK
TITLE = Daten für Takt in temporäre Variablen laden
      A     #in_Anlage_ein;	// (015)
      A     #in_Ansteuerung_Ventil;
      A     DIX [AR2,P#3.6];	// Freigabe Takt (Struktur)
      =     #Freigabe_Takt;
      A     DIX [AR2,P#3.2];	// Start mit Impuls (Struktur)
      =     #Start_mit_Impuls;
      A     DIX [AR2,P#3.3];	// Taktanzahl erreicht (Struktur)
      =     #Taktanzahl_erreicht;
      A     DIX [AR2,P#3.4];	// Dauertakt (Struktur)
      =     #Dauertakt;
      A     DIX [AR2,P#3.7];	// Taktausgang (Struktur)
      =     #Taktausgang;
      L     DID [AR2,P#8.0];	// Impulszeit (Struktur)
      T     #Impulszeit;
      L     DID [AR2,P#12.0];	// Pausezeit (Struktur)
      T     #Pausezeit;
      L     DID [AR2,P#16.0];	// Impuls-/Pausezähler (Struktur)
      T     #Zeitzaehler;
      L     DIW [AR2,P#20.0];	// Sollanzahl Takte (Struktur)
      T     #Sollanzahl_Takte;
      L     DIW [AR2,P#22.0];	// Taktzähler (Struktur)
      T     #Taktzaehler;
NETWORK
TITLE = Rückmeldung für Takt
      A(;
      L     #in_Ventil_Typ;
      L     0;
      ==I;
      );
      A     #io_Ausgang_Ventil;
      O;
      A(;
      L     #in_Ventil_Typ;
      L     1;
      ==I;
      );
      A     #in_Eingang_angesteuert;
      O;
      A(;
      L     #in_Ventil_Typ;
      L     2;
      ==I;
      );
      A     #in_Eingang_angesteuert;
      O;
      A(;
      L     #in_Ventil_Typ;
      L     3;
      ==I;
      );
      AN    #in_Eingang_nicht_angest;
      =     #Rueckmeldung;
NETWORK
TITLE = Takt generieren
      CALL  FC 2 (
           in_Freigabe              := #Freigabe_Takt,
           in_Rueckmeldung          := #Rueckmeldung,
           in_Start_mit_Impuls      := #Start_mit_Impuls,
           in_Dauertakt             := #Dauertakt,
           in_Impuls                := M 1.7,
           in_Impulszeit_in_100ms   := MW 6,
           in_Impulszeit            := #Impulszeit,
           in_Pausezeit             := #Pausezeit,
           in_Sollanzahl_Takte      := #Sollanzahl_Takte,
           io_Taktausgang           := #Taktausgang,
           io_Taktanzahl_erreicht   := #Taktanzahl_erreicht,
           io_Zeitzaehler           := #Zeitzaehler,
           io_Taktzaehler           := #Taktzaehler);
NETWORK
TITLE = Ansteuerung Ventil
      A     #in_Anlage_ein;	// (015)
      A(;
      ON    #in_Quitt_Stoerung_noetig;
      O;
      A     #in_Quitt_Stoerung_noetig;
      AN    #io_Stoerung;
      );
      A(;
      AN    DIX [AR2,P#2.6];	// Automatikmode zu Farbgrafik (Struktur)
      AN    DIX [AR2,P#3.6];	// Freigabe Takt (Struktur)
      A     #in_Ansteuerung_Ventil;
      O;
      AN    DIX [AR2,P#2.6];	// Automatikmode zu Farbgrafik (Struktur)
      A     DIX [AR2,P#3.6];	// Freigabe Takt (Struktur)
      A     #Taktausgang;
      O;
      A     DIX [AR2,P#2.6];	// Handmode zu Farbgrafik (Struktur)
      A     DIX [AR2,P#3.0];	// Ansteuerung Handmode von Farbgrafik (Struktur)
      );
      =     #io_Ausgang_Ventil;
NETWORK
TITLE = Ventiltyp festlegen
      L     #in_Ventil_Typ;
      L     0;
      ==I;
      JC    TYP0;	// Sprung zu Ventil Typ 0
      TAK;
      L     1;
      ==I;
      JC    TYP1;	// Sprung zu Ventil Typ 1
      TAK;
      L     2;
      ==I;
      JC    TYP2;	// Sprung zu Ventil Typ 2
      TAK;
      L     3;
      ==I;
      JC    TYP3;	// Sprung zu Ventil Typ 3
      JU    ENDE;
NETWORK
TITLE = Betriebsmeldung Typ 0 (kein Eingang)
TYP0: A     #io_Ausgang_Ventil;
      A(;	// (011)
      L     DIW [AR2,P#40.0];	// (011) Istzeit Verzögerung (Struktur) 
      L     DIW [AR2,P#38.0];	// (011) Sollzeit Verzögerung (Struktur)
      >=I;	// (011)
      );	// (011)
      =     #io_Ventil_in_Betrieb;	// Betriebsmeldung anzeigen
NETWORK
TITLE = Istzähler Verzögerung hochzählen (011)
      A     #io_Ausgang_Ventil;
      AN    M 4.5;	// Sekundenimpuls (Standardmerker)
      O     #io_Ventil_in_Betrieb;	// Betriebsmeldung anzeigen
      JC    KVZ;
      L     DIW [AR2,P#40.0];	// Istzeit Verzögerung (Struktur)
      +     1;
      T     DIW [AR2,P#40.0];	// Istzeit Verzögerung (Struktur)
KVZ:  NOP   0;
NETWORK
TITLE = Istzähler Verzögerung zurücksetzen (011)
      O     #io_Ausgang_Ventil;
      JC    RVZ;
      L     0;
      T     DIW [AR2,P#40.0];	// Istzeit Verzögerung (Struktur)
RVZ:  NOP   0;
NETWORK
TITLE = Diskrepanz Typ 0 (kein Eingang)
      CLR;	// keine Diskrepanz möglich
      =     #Diskrepanz;
      JU    STOE;
NETWORK
TITLE = Betriebsmeldung Typ1 (Eingang angesteuert und nicht angesteuert)
TYP1: A     #io_Ausgang_Ventil;
      A     #in_Eingang_angesteuert;
      AN    #in_Eingang_nicht_angest;
      =     #io_Ventil_in_Betrieb;
NETWORK
TITLE = Diskrepanz Typ 1 (Eingang angesteuert und nicht angesteuert)
      A     #io_Ausgang_Ventil;
      AN    #in_Eingang_angesteuert;
      O;
      AN    #io_Ausgang_Ventil;
      AN    #in_Eingang_nicht_angest;
      O;
      A     #in_Eingang_angesteuert;
      A     #in_Eingang_nicht_angest;
      O;
      AN    #in_Eingang_angesteuert;
      AN    #in_Eingang_nicht_angest;
      =     #Diskrepanz;
      JU    STOE;
NETWORK
TITLE = Betriebsmeldung Typ 2 (Eingang angesteuert)
TYP2: A     #io_Ausgang_Ventil;
      A     #in_Eingang_angesteuert;
      =     #io_Ventil_in_Betrieb;
NETWORK
TITLE = Diskrepanz Typ 2 (Eingang angesteuert)
      A     #io_Ausgang_Ventil;
      AN    #in_Eingang_angesteuert;
      O;
      AN    #io_Ausgang_Ventil;
      A     #in_Eingang_angesteuert;
      =     #Diskrepanz;
      JU    STOE;
NETWORK
TITLE = Betriebsmeldung Typ 3 (Eingang nicht angesteuert)
TYP3: A     #io_Ausgang_Ventil;
      AN    #in_Eingang_nicht_angest;
      =     #io_Ventil_in_Betrieb;
NETWORK
TITLE = Diskrepanz Typ 3 (Eingang nicht angesteuert)
      A     #io_Ausgang_Ventil;
      A     #in_Eingang_nicht_angest;
      O;
      AN    #io_Ausgang_Ventil;
      AN    #in_Eingang_nicht_angest;
      =     #Diskrepanz;
NETWORK
TITLE = Störungszähler
STOE: A     #in_Quitt_Stoerung_noetig;
      AN    #in_Quitt_Stoerung;
      A     #io_Stoerung;
      O;
      A     #Diskrepanz;
      AN    #in_Quitt_Stoerung;	// (008)
      O;	// (008)
      AN    #in_Quitt_Stoerung_noetig;	// (008)
      A     #Diskrepanz;	// (008)
      JC    SZ1;
      L     0;	// Wenn keine Diskrepanz dann Zähler löschen
      T     DIW [AR2,P#6.0];	// Istzeit Störung (Struktur)
      JU    ESZ;
// Störungszähler in jeder Sekunde erhöhen
SZ1:  O     #io_Stoerung;
      ON    M 4.5;	// Sekundenimpuls (Standardmerker)
      JC    ESZ;
      L     DIW [AR2,P#6.0];	// Istzeit Störung (Struktur)
      +     1;	// (012)
      T     DIW [AR2,P#6.0];	// Istzeit Störung (Struktur)
ESZ:  NOP   0;
NETWORK
TITLE = Störmeldung ausgeben
      L     DIW [AR2,P#6.0];	// Istzeit Störung (Struktur)
      L     DIW [AR2,P#4.0];	// Sollzeit Störung (Struktur)
      >=I;
      =     #io_Stoerung;
NETWORK
TITLE = Stoerung quittieren
      O     #Diskrepanz;	// Stoerung steht noch an
      ON    #io_Stoerung;
      JC    ESQ;
      ON    #in_Quitt_Stoerung_noetig;	// Stoerung muß quittiert werden ?
      JC    SQ1;	// Stoerung muß nicht quittiert werden
      A     #in_Quitt_Stoerung;
SQ1:  R     #io_Stoerung;
ESQ:  NOP   0;
NETWORK
TITLE = Flankenauswertung Ausgang Ventil für Schalthäufigkeitzähler
      A     #io_Ausgang_Ventil;
      FP    DIX [AR2,P#24.3];	// Flankenmerker Ausgang (Struktur)
      =     #positive_Flanke;
NETWORK
TITLE = Schalthäufigkeitzähler
      ON    DIX [AR2,P#0.3];	// Kennung Schalthäufigkeitzähler ein (Struktur)
      ON    #positive_Flanke;
      JC    ESHZ;
      L     1.000000e+00;
      L     DID [AR2,P#26.0];	// Schalthäufigkeitzähler (Struktur)
      +R;
      T     DID [AR2,P#26.0];	// Schalthäufigkeitzähler (Struktur)
ESHZ: NOP   0;
NETWORK
TITLE = Schalthäufigkeitzähler zurücksetzten
      AN    DIX [AR2,P#24.0];	// Reset Schalthäufigkeitzähler (Struktur)
      JC    E_RS;
      L     0.000000e+00;
      T     DID [AR2,P#26.0];	// Schalthäufigkeitzähler (Struktur)
      CLR;
      =     DIX [AR2,P#24.0];	// Reset Schalthäufigkeitzähler (Struktur)
E_RS: NOP   0;
NETWORK
TITLE = Warnmeldung Schalthäufigkeitszähler erzeugen
      A(;
      L     DID [AR2,P#26.0];	// Schalthäufigkeitzähler (Struktur)
      L     DID [AR2,P#30.0];	// Sollwert Warnung (Struktur)
      >R;
      );
      A(;
      L     DID [AR2,P#30.0];	// Sollwert Warnung (Struktur)
      L     0.000000e+00;
      <>R;
      );
      =     DIX [AR2,P#24.1];	// Warnmeldung Schalthäufigkeitzähler (Struktur)
NETWORK
TITLE = Alarmmeldung Schalthäufigkeitszähler erzeugen
      A(;
      L     DID [AR2,P#26.0];	// Schalthäufigkeitzähler (Struktur)
      L     DID [AR2,P#34.0];	// Sollwert Alarm (Struktur)
      >R;
      );
      A(;
      L     DID [AR2,P#34.0];	// Sollwert Alarm (Struktur)
      L     0.000000e+00;
      <>R;
      );
      =     DIX [AR2,P#24.2];	// Alarmmeldung Schalthäufigkeitzähler (Struktur)
NETWORK
TITLE =  Objektstatus für Visualisation OP (009) (010)
//Stati:
//-------
//1 = nicht in Betrieb, keine Störung ==> Farbvorschlag weiß
//5 = angesteuert, in Betrieb, keine Störung ==> Farbvorschlag grün
//9 = angesteuert, nicht in Betrieb, keine Störung ==> Farbvorschlag grau
//16 = Störung ==> Farbvorschlag rot
// 1 = nicht in Betrieb, keine Störung ==> Farbvorschlag weiß
      L     1;
      AN    #io_Ausgang_Ventil;
      AN    #io_Stoerung;
      AN    DIX [AR2,P#1.3];	// (014) Kennung "invers"
      O;
      A     #io_Ausgang_Ventil;
      A     #io_Ventil_in_Betrieb;
      AN    #io_Stoerung;
      A     DIX [AR2,P#1.3];	// (014) Kennung "invers"
      JC    disp;
// 5 = angesteuert, in Betrieb, keine Störung ==> Farbvorschlag grün
      L     5;
      A     #io_Ausgang_Ventil;
      A     #io_Ventil_in_Betrieb;
      AN    #io_Stoerung;
      AN    DIX [AR2,P#1.3];	// (014) Kennung "invers"
      O;
      AN    #io_Ausgang_Ventil;
      AN    #io_Stoerung;
      A     DIX [AR2,P#1.3];	// (014) Kennung "invers"
      JC    disp;
// 9 = angesteuert, nicht in Betrieb, keine Störung ==> Farbvorschlag grau
      L     9;
      A     #io_Ausgang_Ventil;
      AN    #io_Ventil_in_Betrieb;
      AN    #io_Stoerung;
      JC    disp;
// 16 = Störung ==> Farbvorschlag rot
      L     16;
      A     #io_Stoerung;
      JC    disp;
      L     0;
disp: T     #Objektstatus;
NETWORK
TITLE = Daten in Struktur speichern
      A     #in_Anlage_ein;	// (015)
      =     DIX [AR2,P#42.0];	// (015) Anlage ein (Struktur)
      A     #in_Eingang_angesteuert;
      =     DIX [AR2,P#2.1];	// Eingang angesteuert (Struktur)
      A     #in_Eingang_nicht_angest;
      =     DIX [AR2,P#2.2];	// Eingang nicht angesteuert (Struktur)
      A     #io_Ausgang_Ventil;
      =     DIX [AR2,P#2.0];	// Ausgang Ventil (Struktur)
      A     #io_Ventil_in_Betrieb;
      =     DIX [AR2,P#2.4];	// Ventil in Betrieb (Struktur)
      A     #io_Stoerung;
      =     DIX [AR2,P#2.5];	// Störung (Struktur)
      A     #Taktanzahl_erreicht;
      =     DIX [AR2,P#3.3];	// Taktanzahl erreicht (Struktur)
      A     #Taktausgang;
      =     DIX [AR2,P#3.7];	// Taktausgang (Struktur)
      L     #Zeitzaehler;
      T     DID [AR2,P#16.0];	// Impuls-/Pausezähler (Struktur)
      L     #Taktzaehler;
      T     DIW [AR2,P#22.0];	// Taktzähler (Struktur)
      L     #Objektstatus;	// (009)
      T     DIW [AR2,P#48.0];	// #Objektstatus  (Struktur)   // (009)
NETWORK
TITLE = ENDE
ENDE: NOP   0;
END_FUNCTION

FUNCTION FC 22 : VOID
TITLE = Block for valve actuation and fault monitoring 2O,2I
//Erstellung:
//Datum        Bearbeiter                                                 Version
//--------------------------------------------------------------------------------
//24.09.98     A.Geiger (gea)                                             01.00.00
//
//Änderungen:
//Nr. Datum    Bearb Änderung                                       Marke  Version
//--------------------------------------------------------------------------------
//01  16.04.99 sra   Fehlerbeseitigung Störungsquittierung          ()    01.00.01
//02  21.05.99 sra   Einfügen der Handbedienuung                    ()    01.01.00
//03  23.07.99 sra   Ausg. wird auch bei Simulation gesetzt         ()    01.01.01
//04  19.10.99 sra   Anpassung an neue Struktur                     ()    01.02.00
//05  19.09.00 sra   komplette Überarbeitung / neue Struktur        ()    02.00.00
//06  15.02.01 sra   Rücksetzen Istwert Störung bei Quitt.          ()    02.00.01
//07  31.03.03 sra   Fehlerbeseitigung Störungsquittierung          (007) 02.00.02
//08  23.03.05 sra   Änderung Störungsquittierung                   (008) 02.01.00
//09  31.10.05 sra   Ansteuerung Handbedienung im Automode rücksetz.
//                   Handbedienung zentral sperren                  (009) 02.02.00
//10  03.05.06 gea   Fehlerbeseitigung Störungszähler               (010) 02.02.01
//11  18.02.09 kmj   Objektstatus ergänzt                           (011) 02.03.00
//12  20.03.09 kal   Objektstatus ergänzt (überarbeitet)            (012) 02.03.01
//13  24.04.09 gea   Handmode zurücksetzen wenn Handmode gesperrt   (013) 02.03.02
//14  10.09.09 sra   Objektststatus für OP ergänzt (erweitert)      (014) 02.04.00
//15  15.10.09 gea   Korrektur Taktpause                            (015) 02.04.01
//16  26.03.12 jm    Objektstatus korrigiert                        (016) 02.04.02
//17  07.09.12 jm    Ohjektstatus aufgeteilt (3 Versionen)          (017) 02.04.03
//18  12.10.12 jm    Objektstatus 3 optimiert                       (018) 02.04.04
//19  15.10.12 jm    Objektstatus 3 optimiert (1,6 anstatt 1,5)     (019) 02.04.05
//20  18.12.12 sra   Kennung links rechts eingefügt                 (020) 02.05.00
//21  05.12.13 sra   "Anlage ein" eingefügt (Not-Aus-Konzept)       (021) 02.06.00
//22  24.07.14 jm    Ohjektstatus ergänzt/geändert                  (022) 02.07.01
//23  09.03.16 jm    Objektstatus 9/19 bis Ende oder Störung        (023) 02.07.02
//________________________________________________________________________________
//Funktion:
//
//-Der Baustein steuert den Ablauf eines Ventils mit 2 Ausgängen und 2 Eingängen.
//
//-Die Ausgänge werden nur angesteuert wenn der Eingang "in_Anlage_ein" = true
// ist. Diese Funktion ist vorhanden, um bei einem Not-Halt die Anlage vor 
// unkontrolliertem Einschalten zu schützen. 
//
//-Ist in der Ventilstruktur die Taktfunktion freigegeben wird bei Freigabe des 
// Ventils der Ausgang entsprechend der Impuls-/Pausezeit angesteuert.
//
//-Der Baustein überwacht den Zustand der Ausgänge und der Eingänge und generiert 
// nach Ablauf der "Sollzeit Störung" eine Störmeldung
//
//-Ist das Bit "Simulation" auf TRUE, so werden die Eingänge simuliert.
//
//-Ist die Kennung "Schalthäufigkeitszähler_ein" aktiviert werden die
// Ansteuerungen des Ventils aufsummiert. Dies erfolgt mit setzen des Ausgangs.
//
//-Der Baustein kopiert die Parameter "in_Eingang_...", "io_Ausgang_...", 
// "in_Quitt_Stoerung" und "io_Stoerung" in die angegebene Datenstruktur zur 
// Visualisierung auf einem Farbgrafiksystem. Diese Parameter müssen folglich 
// nicht mehr extern umkopiert werden.
//
//-Ist der Parameter "in_Handbedienung_erlaubt" angewählt kann das Ventil über 
// eine Farbgrafik oder ein Bedienterminal manuell angesteuert werden
//
AUTHOR : gea
FAMILY : AZO
NAME : standard
VERSION : 0.0
VAR_INPUT
  in_Handbedienung_erlaubt : BOOL ;	//1 = manual operation permitted, 0 = manual operation not permitted/locked
  in_Quitt_Stoerung_noetig : BOOL ;	//1 = fault acknowledgement required, 0 = automatic fault acknowledgement
  in_Quitt_Stoerung : BOOL ;	//Fault acknowledgement when fault_acknowledgement_required = 1
  in_Anlage_ein : BOOL ;	//Anlage bzw. Anlagenbereich nach Not-Halt freigegeben
  in_Ansteuerung_Stellung1 : BOOL ;	//Actuation of valve position 1 in automatic mode
  in_Ansteuerung_Stellung2 : BOOL ;	//Actuation of valve position 2 in automatic mode
  in_Eingang_Stellung_1 : BOOL ;	//Valve intake when position 1 actuated
  in_Eingang_Stellung_2 : BOOL ;	//Valve intake when position 2 actuated
END_VAR
VAR_IN_OUT
  io_Ausgang_Stellung_1 : BOOL ;	//Valve output to actuate position 1
  io_Ausgang_Stellung_2 : BOOL ;	//Valve output to actuate position 2
  io_Stellung_1_Betrieb : BOOL ;	//Signal "position 1 in operation" (position 1 actuated)
  io_Stellung_2_Betrieb : BOOL ;	//Signal "position 2 in operation" (position 2 actuated)
  io_Stoerung : BOOL ;	//Signal "valve fault"
  io_Ventilstruktur : ANY ;	//ANY pointer of valve structure
END_VAR
VAR_TEMP
  Freigabe_Takt : BOOL ;
  Rueckmeldung : BOOL ;
  Start_mit_Impuls : BOOL ;
  Dauertakt : BOOL ;
  Taktausgang : BOOL ;
  Taktanzahl_erreicht : BOOL ;
  Diskrepanz : BOOL ;
  positive_Flanke : BOOL ;
  Impulszeit : REAL ;
  Pausezeit : REAL ;
  Sollanzahl_Takte : INT ;
  Zeitzaehler : REAL ;
  Taktzaehler : INT ;
  Objektstatus : INT ;
END_VAR
BEGIN
NETWORK
TITLE = Anfangs-DW der Struktur aus ANY-Zeiger auslesen
      L     P##io_Ventilstruktur;
      LAR2;
      L     D [AR2,P#6.0];
      LAR2;
NETWORK
TITLE = Simulation
      AN    DIX [AR2,P#4.1];	// Simulation ein (Struktur)
      JC    ESIM;
      A     #io_Ausgang_Stellung_1;
      AN    #io_Ausgang_Stellung_2;
      O;
      AN    #io_Ausgang_Stellung_2;
      AN    DIX [AR2,P#2.2];	// Eingang Stellung 1 (Struktur)
      AN    DIX [AR2,P#2.3];	// Eingang Stellung 2 (Struktur)
      O;
      AN    #io_Ausgang_Stellung_1;
      AN    #io_Ausgang_Stellung_2;
      A     DIX [AR2,P#2.2];	// Eingang Stellung 1 (Struktur)
      S     #in_Eingang_Stellung_1;
      R     #in_Eingang_Stellung_2;
      AN    #io_Ausgang_Stellung_1;
      A     #io_Ausgang_Stellung_2;
      O;
      AN    #io_Ausgang_Stellung_1;
      AN    #io_Ausgang_Stellung_2;
      A     DIX [AR2,P#2.3];	// Eingang Stellung 2 (Struktur)
      R     #in_Eingang_Stellung_1;
      S     #in_Eingang_Stellung_2;
ESIM: NOP   0;
NETWORK
TITLE = Umschaltung Hand-/Automatikmode 
      A     DIX [AR2,P#3.2];	// Handmode von Farbgrafik (Struktur)
      AN    DIX [AR2,P#3.5];	// Handmode gesperrt (Struktur)
      AN    M 0.0;	// Handbedienung zentral sperren (009)
      S     DIX [AR2,P#3.1];	// Handmode zu Farbgrafik (Struktur)
      ON    DIX [AR2,P#3.2];	// Handmode von Farbgrafik (Struktur)
      ON    #in_Handbedienung_erlaubt;
      O     M 0.0;	// Handbedienung zentral sperren (009)
      O     DIX [AR2,P#3.5];	// Handmode gesperrt (Struktur) (013)
      R     DIX [AR2,P#3.1];	// Handmode zu Farbgrafik (Struktur)
      R     DIX [AR2,P#3.2];	// Handmode von Farbgrafik (Struktur) (009)
NETWORK
TITLE = Ansteuerung Handmode zurücksetzen
//(009) 
      AN    DIX [AR2,P#3.1];	// Handmode zu Farbgrafik (Struktur)
      R     DIX [AR2,P#3.3];	// Ansteuerung Stellung 1 Handmode von Farbgrafik (Struktur)
      R     DIX [AR2,P#3.4];	// Ansteuerung Stellung 2 Handmode von Farbgrafik (Struktur)
NETWORK
TITLE = Daten für Takt in temporäre Variablen laden
      A     #in_Anlage_ein;	// (021)
      A(;
      O     #in_Ansteuerung_Stellung1;
      O     #in_Ansteuerung_Stellung2;
      );
      A     DIX [AR2,P#4.2];	// Freigabe Takt (Struktur)
      =     #Freigabe_Takt;
      A     DIX [AR2,P#3.6];	// Start mit Impuls (Struktur)
      =     #Start_mit_Impuls;
      A     DIX [AR2,P#3.7];	// Taktanzahl erreicht (Struktur)
      =     #Taktanzahl_erreicht;
      A     DIX [AR2,P#4.0];	// Dauertakt (Struktur)
      =     #Dauertakt;
      A     DIX [AR2,P#4.3];	// Taktausgang (Struktur)
      =     #Taktausgang;
      L     DID [AR2,P#10.0];	// Impulszeit (Struktur)
      T     #Impulszeit;
      L     DID [AR2,P#14.0];	// Pausezeit (Struktur)
      T     #Pausezeit;
      L     DID [AR2,P#18.0];	// Impuls-/Pausezähler (Struktur)
      T     #Zeitzaehler;
      L     DIW [AR2,P#22.0];	// Sollanzahl Takte (Struktur)
      T     #Sollanzahl_Takte;
      L     DIW [AR2,P#24.0];	// Taktzähler (Struktur)
      T     #Taktzaehler;
NETWORK
TITLE = Rückmeldung für Takt
// (network holds code this reader does not know; not shown)
NETWORK
TITLE = Takt generieren
      CALL  FC 2 (
           in_Freigabe              := #Freigabe_Takt,
           in_Rueckmeldung          := #Rueckmeldung,
           in_Start_mit_Impuls      := #Start_mit_Impuls,
           in_Dauertakt             := #Dauertakt,
           in_Impuls                := M 1.7,
           in_Impulszeit_in_100ms   := MW 6,
           in_Impulszeit            := #Impulszeit,
           in_Pausezeit             := #Pausezeit,
           in_Sollanzahl_Takte      := #Sollanzahl_Takte,
           io_Taktausgang           := #Taktausgang,
           io_Taktanzahl_erreicht   := #Taktanzahl_erreicht,
           io_Zeitzaehler           := #Zeitzaehler,
           io_Taktzaehler           := #Taktzaehler);
NETWORK
TITLE = Ansteuerung Stellung 1
      A     #in_Anlage_ein;	// (021)
      A(;
      ON    #in_Quitt_Stoerung_noetig;
      O;
      A     #in_Quitt_Stoerung_noetig;
      AN    #io_Stoerung;
      );
      A(;
      AN    DIX [AR2,P#3.1];	// Automatikmode zu Farbgrafik (Struktur)
      AN    DIX [AR2,P#4.2];	// Freigabe Takt (Struktur)
      A     #in_Ansteuerung_Stellung1;
      AN    #in_Ansteuerung_Stellung2;
      O;
      AN    DIX [AR2,P#3.1];	// Automatikmode zu Farbgrafik (Struktur)
      A     DIX [AR2,P#4.2];	// Freigabe Takt (Struktur)
      A     #Taktausgang;
      O;
      A     DIX [AR2,P#3.1];	// Handmode zu Farbgrafik (Struktur)
      A     DIX [AR2,P#3.3];	// Ansteuerung Stellung 1 Handmode von Farbgrafik (Struktur)
      AN    DIX [AR2,P#3.4];	// Ansteuerung Stellung 2 Handmode von Farbgrafik (Struktur)
      );
      =     #io_Ausgang_Stellung_1;
NETWORK
TITLE = Ansteuerung Stellung 2
      A     #in_Anlage_ein;	// (021)
      A(;
      ON    #in_Quitt_Stoerung_noetig;
      O;
      A     #in_Quitt_Stoerung_noetig;
      AN    #io_Stoerung;
      );
      A(;
      AN    DIX [AR2,P#3.1];	// Automatikmode zu Farbgrafik (Struktur)
      AN    DIX [AR2,P#4.2];	// Freigabe Takt (Struktur)
      A     #in_Ansteuerung_Stellung2;
      AN    #in_Ansteuerung_Stellung1;
      O;
      AN    DIX [AR2,P#3.1];	// Automatikmode zu Farbgrafik (Struktur)
      A     DIX [AR2,P#4.2];	// Freigabe Takt (Struktur)
      AN    #Taktausgang;
      O;
      A     DIX [AR2,P#3.1];	// Handmode zu Farbgrafik (Struktur)
      AN    DIX [AR2,P#3.3];	// Ansteuerung Stellung 1 Handmode von Farbgrafik (Struktur)
      A     DIX [AR2,P#3.4];	// Ansteuerung Stellung 2 Handmode von Farbgrafik (Struktur)
      );
      =     #io_Ausgang_Stellung_2;
NETWORK
TITLE = Betriebsmeldung Stellung 1
      A     #io_Ausgang_Stellung_1;
      A     #in_Eingang_Stellung_1;
      AN    #io_Ausgang_Stellung_2;
      AN    #in_Eingang_Stellung_2;
      =     #io_Stellung_1_Betrieb;
NETWORK
TITLE = Betriebsmeldung Stellung 2
      AN    #io_Ausgang_Stellung_1;
      AN    #in_Eingang_Stellung_1;
      A     #io_Ausgang_Stellung_2;
      A     #in_Eingang_Stellung_2;
      =     #io_Stellung_2_Betrieb;
NETWORK
TITLE = Diskrepanz
      A     #io_Ausgang_Stellung_1;	// Nicht auf Abzweig
      AN    #in_Eingang_Stellung_1;
      O;
      A     #io_Ausgang_Stellung_2;	// Nicht auf Gerade
      AN    #in_Eingang_Stellung_2;
      O;
      A     #in_Eingang_Stellung_1;	// Stellung nicht definiert
      A     #in_Eingang_Stellung_2;
      O;
      AN    #in_Eingang_Stellung_1;	// Stellung nicht definiert
      AN    #in_Eingang_Stellung_2;
      O;
      A     #in_Ansteuerung_Stellung1;	// Ansteuerung nicht zulässig
      A     #in_Ansteuerung_Stellung2;
      =     #Diskrepanz;	// Diskrepanz feststellen
NETWORK
TITLE = Störungszähler
      A     #in_Quitt_Stoerung_noetig;
      AN    #in_Quitt_Stoerung;
//      U     #Diskrepanz                 // (007)
      A     #io_Stoerung;
      O;
//      UN    #in_Quitt_Stoerung_noetig   // (007)
      A     #Diskrepanz;
      AN    #in_Quitt_Stoerung;	// (008)
      O;	// (010)
      AN    #in_Quitt_Stoerung_noetig;	// (010)
      A     #Diskrepanz;	// (010)
      JC    SZ1;
      L     0;	// Wenn keine Diskrepanz dann Zähler löschen
      T     DIW [AR2,P#8.0];	// Istzeit Störung (Struktur)
      JU    ESZ;
// Störungszähler in jeder Sekunde erhöhen
SZ1:  O     #io_Stoerung;
      ON    M 4.5;	// Sekundenimpuls (Standardmerker)
      JC    ESZ;
      L     DIW [AR2,P#8.0];	// Istzeit Störung (Struktur)
      INC   1;
      T     DIW [AR2,P#8.0];	// Istzeit Störung (Struktur)
ESZ:  NOP   0;
NETWORK
TITLE = Störmeldung ausgeben
      L     DIW [AR2,P#8.0];	// Istzeit Störung (Struktur)
      L     DIW [AR2,P#6.0];	// Sollzeit Störung (Struktur)
      >=I;
      =     #io_Stoerung;
NETWORK
TITLE = Stoerung quittieren
      O     #Diskrepanz;	// Stoerung steht noch an
      ON    #io_Stoerung;
      JC    ESQ;
      ON    #in_Quitt_Stoerung_noetig;	// Stoerung muß quittiert werden ?
      JC    SQ1;	// Stoerung muß nicht quittiert werden
      A     #in_Quitt_Stoerung;
SQ1:  R     #io_Stoerung;
ESQ:  NOP   0;
NETWORK
TITLE = Flankenauswertung Ausgang Ventil für Schalthäufigkeitzähler
//Es wird die Schalthäufigkeit der Ventile gezählt !  
      A     #io_Ausgang_Stellung_1;
      A     #in_Eingang_Stellung_1;
      O;
      A     #io_Ausgang_Stellung_2;
      A     #in_Eingang_Stellung_2;
      FP    DIX [AR2,P#26.3];	// Flankenmerker Ausgang (Struktur)
      =     #positive_Flanke;
NETWORK
TITLE = Schalthäufigkeitzähler
      ON    DIX [AR2,P#0.3];	// Kennung Schalthäufigkeitzähler ein (Struktur)
      ON    #positive_Flanke;
      JC    ESHZ;
      L     1.000000e+00;
      L     DID [AR2,P#28.0];	// Schalthäufigkeitzähler (Struktur)
      +R;
      T     DID [AR2,P#28.0];	// Schalthäufigkeitzähler (Struktur)
ESHZ: NOP   0;
NETWORK
TITLE = Schalthäufigkeitzähler zurücksetzten
      AN    DIX [AR2,P#26.0];	// Reset Schalthäufigkeitzähler (Struktur)
      JC    E_RS;
      L     0.000000e+00;
      T     DID [AR2,P#28.0];	// Schalthäufigkeitzähler (Struktur)
      CLR;
      =     DIX [AR2,P#26.0];	// Reset Schalthäufigkeitzähler (Struktur)
E_RS: NOP   0;
NETWORK
TITLE = Warnmeldung Schalthäufigkeitzähler erzeugen
      A(;
      L     DID [AR2,P#28.0];	// Schalthäufigkeitzähler (Struktur)
      L     DID [AR2,P#32.0];	// Sollwert Warnung (Struktur)
      >R;
      );
      A(;
      L     DID [AR2,P#32.0];	// Sollwert Warnung (Struktur)
      L     0.000000e+00;
      <>R;
      );
      =     DIX [AR2,P#26.1];	// Warnmeldung Schalthäufigkeitzähler (Struktur)
NETWORK
TITLE = Alarmmeldung Schalthäufigkeitzähler erzeugen
      A(;
      L     DID [AR2,P#28.0];	// Schalthäufigkeitzähler (Struktur)
      L     DID [AR2,P#36.0];	// Sollwert Alarm (Struktur)
      >R;
      );
      A(;
      L     DID [AR2,P#36.0];	// Sollwert Alarm (Struktur)
      L     0.000000e+00;
      <>R;
      );
      =     DIX [AR2,P#26.2];	// Alarmmeldung Schalthäufigkeitzähler (Struktur)
NETWORK
TITLE = Objektstatus für Visualisation OP (011)(012)(017)
//Stati:
//-------
//1 = nicht angesteuert, Ventil in Position 1, keine Störung ==> grau
//2 = nicht angesteuert, Ventil in Position 2, keine Störung ==> grau
//5 = Position 1 angesteuert, Ventil in Position 1, keine Störung ==> grün
//6 = Position 2 angesteuert, Ventil in Position 2, keine Störung ==> grün
//9 = Position 1 angesteuert, Ventil nicht in Position 1, keine Störung ==> weiß
//10 = Position 2 angesteuert, Ventil nicht in Position 2, keine Störung ==> weiß
//14 = Störung, quittierpflichtig, Ausgang nicht angesteuert, Störung ==> rot/weiß
//15 = Störung, nicht quittierpflichtig, Ausgang angesteuert, Störung ==> rot/grün
//16 = Störung quittiert ==> rot
      A(;
      O     DIX [AR2,P#0.7];	// Kennung "gerade/abzweig"
      O     DIX [AR2,P#1.0];	// Kennung "Stellung1/Stellung2"
      O     DIX [AR2,P#1.6];	// Kennung "links/rechts"               (020)
      );
      JCN   NSV1;	// Not Status Version 1
// 1 ==> grau
      L     1;
      AN    #io_Stoerung;
      A(;
      AN    DIX [AR2,P#0.5];	// Kennung "invers"
      A     #in_Eingang_Stellung_1;
      AN    #in_Eingang_Stellung_2;
      AN    #io_Ausgang_Stellung_1;
      AN    #io_Ausgang_Stellung_2;
      O;
      A     DIX [AR2,P#0.5];	// Kennung "invers"
      AN    #in_Eingang_Stellung_1;
      A     #in_Eingang_Stellung_2;
      AN    #io_Ausgang_Stellung_1;
      AN    #io_Ausgang_Stellung_2;
      );
      JC    disp;
// 2 ==> grau
      L     2;
      AN    #io_Stoerung;
      A(;
      AN    DIX [AR2,P#0.5];	// Kennung "invers"
      AN    #in_Eingang_Stellung_1;
      A     #in_Eingang_Stellung_2;
      AN    #io_Ausgang_Stellung_1;
      AN    #io_Ausgang_Stellung_2;
      O;
      A     DIX [AR2,P#0.5];	// Kennung "invers"
      A     #in_Eingang_Stellung_1;
      AN    #in_Eingang_Stellung_2;
      AN    #io_Ausgang_Stellung_1;
      AN    #io_Ausgang_Stellung_2;
      );
      JC    disp;
// 5 ==> grün
      L     5;
      AN    #io_Stoerung;
      A(;
      AN    DIX [AR2,P#0.5];	// Kennung "invers"
      A     #in_Eingang_Stellung_1;
      AN    #in_Eingang_Stellung_2;
      A     #io_Ausgang_Stellung_1;
      AN    #io_Ausgang_Stellung_2;
      O;
      A     DIX [AR2,P#0.5];	// Kennung "invers"
      AN    #in_Eingang_Stellung_1;
      A     #in_Eingang_Stellung_2;
      AN    #io_Ausgang_Stellung_1;
      A     #io_Ausgang_Stellung_2;
      );
      JC    disp;
// 6 ==> grün
      L     6;
      AN    #io_Stoerung;
      A(;
      AN    DIX [AR2,P#0.5];	// Kennung "invers"
      AN    #in_Eingang_Stellung_1;
      A     #in_Eingang_Stellung_2;
      AN    #io_Ausgang_Stellung_1;
      A     #io_Ausgang_Stellung_2;
      O;
      A     DIX [AR2,P#0.5];	// Kennung "invers"
      A     #in_Eingang_Stellung_1;
      AN    #in_Eingang_Stellung_2;
      A     #io_Ausgang_Stellung_1;
      AN    #io_Ausgang_Stellung_2;
      );
      JC    disp;
// 9 ==> weiß
      L     9;
      AN    #io_Stoerung;
      A(;
      AN    DIX [AR2,P#0.5];	// Kennung "invers"
      AN    #in_Eingang_Stellung_1;
//      UN    #in_Eingang_Stellung_2    // (023)
      A     #io_Ausgang_Stellung_1;
      AN    #io_Ausgang_Stellung_2;
      O;
      A     DIX [AR2,P#0.5];	// Kennung "invers"
//      UN    #in_Eingang_Stellung_1    // (023)
      AN    #in_Eingang_Stellung_2;
      AN    #io_Ausgang_Stellung_1;
      A     #io_Ausgang_Stellung_2;
      );
      JC    disp;
// 10 ==> weiß
      L     10;
      AN    #io_Stoerung;
      A(;
      AN    DIX [AR2,P#0.5];	// Kennung "invers"
//      UN    #in_Eingang_Stellung_1    // (023)
      AN    #in_Eingang_Stellung_2;
      AN    #io_Ausgang_Stellung_1;
      A     #io_Ausgang_Stellung_2;
      O;
      A     DIX [AR2,P#0.5];	// Kennung "invers"
      AN    #in_Eingang_Stellung_1;
//      UN    #in_Eingang_Stellung_2    // (023)
      A     #io_Ausgang_Stellung_1;
      AN    #io_Ausgang_Stellung_2;
      );
      JC    disp;
// 14 = Störung, quittierpflichtig, Ausgang nicht angesteuert, Störung ==> rot/weiß
      L     14;	// (014)
      A     #io_Stoerung;	// (014)
      AN    #in_Quitt_Stoerung;	// (014)
      AN    #io_Ausgang_Stellung_1;	// (014)
      AN    #io_Ausgang_Stellung_2;	// (014)
      JC    disp;	// (014)
// 15 = Störung, nicht quittierpflichtig, Ausgang angesteuert, Störung ==> rot/grün
      L     15;	// (014)
      A     #io_Stoerung;	// (014)
      AN    #in_Quitt_Stoerung;	// (014)
      A(;	// (014)
      O     #io_Ausgang_Stellung_1;	// (014)
      O     #io_Ausgang_Stellung_2;	// (014)
      );	// (014)
      JC    disp;	// (014)
// 16 = Störung quittiert ==> rot
      L     16;
      A     #io_Stoerung;
      JC    disp;
NSV1: NOP   0;
NETWORK
TITLE = Objektstatus für Visualisation OP (011)(012)(017)
//Stati:
//-------
//1 = nicht angesteuert, Ventil in Position 1, keine Störung ==> grau
//2 = nicht angesteuert, Ventil in Position 2, keine Störung ==> grau
//5 = Position 1 angesteuert, Ventil in Position 1, keine Störung ==> grün
//6 = Position 2 angesteuert, Ventil in Position 2, keine Störung ==> grün
//9 = Position 1 angesteuert, Ventil nicht in Position 1, keine Störung ==> weiß
//10 = Position 2 angesteuert, Ventil nicht in Position 2, keine Störung ==> weiß
//14 = Störung, quittierpflichtig, Ausgang nicht angesteuert, Störung ==> rot/weiß
//15 = Störung, nicht quittierpflichtig, Ausgang angesteuert, Störung ==> rot/grün
//16 = Störung quittiert ==> rot
      A(;
//      O     DIX [AR2,P#1.1]             // Kennung "oben/unten" // (022)
      O     DIX [AR2,P#1.2];	// Kennung "grob/fein"
      );
      JCN   NSV2;	// Not Status Version 2
// 1 ==> grau
      L     1;
      AN    #io_Stoerung;
      A(;
      AN    DIX [AR2,P#0.5];	// Kennung "invers"
      AN    #in_Eingang_Stellung_1;
      A     #in_Eingang_Stellung_2;
      AN    #io_Ausgang_Stellung_1;
      AN    #io_Ausgang_Stellung_2;
      O;
      A     DIX [AR2,P#0.5];	// Kennung "invers"
      A     #in_Eingang_Stellung_1;
      AN    #in_Eingang_Stellung_2;
      AN    #io_Ausgang_Stellung_1;
      AN    #io_Ausgang_Stellung_2;
      );
      JC    disp;
// 2 ==> grau
      L     2;
      AN    #io_Stoerung;
      A(;
      AN    DIX [AR2,P#0.5];	// Kennung "invers"
//      UN    #in_Eingang_Stellung_1    // (016)
      A     #in_Eingang_Stellung_1;	// (016)
//      U     #in_Eingang_Stellung_2    // (016)
      AN    #in_Eingang_Stellung_2;	// (016)
      AN    #io_Ausgang_Stellung_1;
//      U     #io_Ausgang_Stellung_2    // (016)
      AN    #io_Ausgang_Stellung_2;	// (016)
      O;
      A     DIX [AR2,P#0.5];	// Kennung "invers"
//      U     #in_Eingang_Stellung_1    // (016)
      AN    #in_Eingang_Stellung_1;	// (016)
//      UN    #in_Eingang_Stellung_2    // (016)
      A     #in_Eingang_Stellung_2;	// (016)
//      U     #io_Ausgang_Stellung_1    // (016)
      AN    #io_Ausgang_Stellung_1;	// (016)
      AN    #io_Ausgang_Stellung_2;
      );
      JC    disp;
// 5 ==> grün
      L     5;
      AN    #io_Stoerung;
      A(;
      AN    DIX [AR2,P#0.5];	// Kennung "invers"
//      U     #in_Eingang_Stellung_1    // (016)
      AN    #in_Eingang_Stellung_1;	// (016)
//      UN    #in_Eingang_Stellung_2    // (016)
      A     #in_Eingang_Stellung_2;	// (016)
      AN    #io_Ausgang_Stellung_1;
//      UN    #io_Ausgang_Stellung_2    // (016)
      A     #io_Ausgang_Stellung_2;	// (016)
      O;
      A     DIX [AR2,P#0.5];	// Kennung "invers"
//      UN    #in_Eingang_Stellung_1    // (016)
      A     #in_Eingang_Stellung_1;	// (016)
//      U     #in_Eingang_Stellung_2    // (016)
      AN    #in_Eingang_Stellung_2;	// (016)
//      UN    #io_Ausgang_Stellung_1    // (016)
      A     #io_Ausgang_Stellung_1;	// (016)
      AN    #io_Ausgang_Stellung_2;
      );
      JC    disp;
// 6 ==> grün
      L     6;
      AN    #io_Stoerung;
      A(;
      AN    DIX [AR2,P#0.5];	// Kennung "invers"
      A     #in_Eingang_Stellung_1;
      AN    #in_Eingang_Stellung_2;
      A     #io_Ausgang_Stellung_1;
      AN    #io_Ausgang_Stellung_2;
      O;
      A     DIX [AR2,P#0.5];	// Kennung "invers"
      AN    #in_Eingang_Stellung_1;
      A     #in_Eingang_Stellung_2;
      AN    #io_Ausgang_Stellung_1;
      A     #io_Ausgang_Stellung_2;
      );
      JC    disp;
// 9 ==> weiß
      L     9;
      AN    #io_Stoerung;
      A(;
      AN    DIX [AR2,P#0.5];	// Kennung "invers"
      AN    #in_Eingang_Stellung_1;
      AN    #in_Eingang_Stellung_2;
      AN    #io_Ausgang_Stellung_1;
      A     #io_Ausgang_Stellung_2;
      O;
      A     DIX [AR2,P#0.5];	// Kennung "invers"
      AN    #in_Eingang_Stellung_1;
      AN    #in_Eingang_Stellung_2;
      A     #io_Ausgang_Stellung_1;
      AN    #io_Ausgang_Stellung_2;
      );
      JC    disp;
// 10 ==> weiß
      L     10;
      AN    #io_Stoerung;
      A(;
      AN    DIX [AR2,P#0.5];	// Kennung "invers"
      AN    #in_Eingang_Stellung_1;
      AN    #in_Eingang_Stellung_2;
      A     #io_Ausgang_Stellung_1;
      AN    #io_Ausgang_Stellung_2;
      O;
      A     DIX [AR2,P#0.5];	// Kennung "invers"
      AN    #in_Eingang_Stellung_1;
      AN    #in_Eingang_Stellung_2;
      AN    #io_Ausgang_Stellung_1;
      A     #io_Ausgang_Stellung_2;
      );
      JC    disp;
// 11 ==> hellgrün
      L     11;
      A     DIX [AR2,P#1.2];	// Kennung "grob/fein"
      A     #io_Ausgang_Stellung_1;
      A     #io_Ausgang_Stellung_2;
      AN    #in_Eingang_Stellung_1;
      AN    #in_Eingang_Stellung_2;
      AN    #io_Stoerung;
      JC    disp;
// 14 = Störung, quittierpflichtig, Ausgang nicht angesteuert, Störung ==> rot/weiß
      L     14;	// (014)
      A     #io_Stoerung;	// (014)
      AN    #in_Quitt_Stoerung;	// (014)
      AN    #io_Ausgang_Stellung_1;	// (014)
      AN    #io_Ausgang_Stellung_2;	// (014)
      JC    disp;	// (014)
// 15 = Störung, nicht quittierpflichtig, Ausgang angesteuert, Störung ==> rot/grün
      L     15;	// (014)
      A     #io_Stoerung;	// (014)
      AN    #in_Quitt_Stoerung;	// (014)
      A(;	// (014)
      O     #io_Ausgang_Stellung_1;	// (014)
      O     #io_Ausgang_Stellung_2;	// (014)
      );	// (014)
      JC    disp;	// (014)
// 16 = Störung quittiert ==> rot
      L     16;
      A     #io_Stoerung;
      JC    disp;
NSV2: NOP   0;
NETWORK
TITLE = Objektstatus für Visualisation OP (011)(012)(017)
//Stati:
//-------
//1 = Eingang Position 2, keine Störung ==> grau
//5 = Eingang Position 1, keine Störung ==> grün
//9 = nicht Eingang 1 und nicht Eingang 2, keine Störung ==> weiß
//14 = Störung, Stellung 2, nicht quittiert ==> rot/weiß
//15 = Störung, Stellung 1, nicht quittiert ==> rot/grün
//16 = Störung quittiert ==> rot
      A(;
      O     DIX [AR2,P#0.6];	// Kennung "auf/zu"
      O     DIX [AR2,P#1.1];	// Kennung "oben/unten" // (022)
      O     DIX [AR2,P#1.3];	// Kennung "ein/aus"
      O     DIX [AR2,P#1.4];	// Kennung "spannen/lösen"
      O     DIX [AR2,P#1.5];	// Kennung "andocken/abdocken"
      O     DIX [AR2,P#1.7];	// Kennung "vor/zurück"   // (022)
      );
      JCN   NSV3;	// Not Status Version 3
// 1 ==> grau
      L     1;
      AN    #io_Stoerung;
      A(;
      AN    DIX [AR2,P#0.5];	// Kennung "invers"
      A     #in_Eingang_Stellung_2;
      O;
      A     DIX [AR2,P#0.5];	// Kennung "invers"
      A     #in_Eingang_Stellung_1;
      );
      JC    disp;
// 6 ==> grün
      L     6;	// (019) = besser weil Fehlertoleranter als 5
      AN    #io_Stoerung;
      A(;
      AN    DIX [AR2,P#0.5];	// Kennung "invers"
      A     #in_Eingang_Stellung_1;
      O;
      A     DIX [AR2,P#0.5];	// Kennung "invers"
      A     #in_Eingang_Stellung_2;
      );
      JC    disp;
// 9 ==> weiß
      L     9;
      AN    #io_Stoerung;
      A(;
      AN    DIX [AR2,P#0.5];	// Kennung "invers"
      AN    #in_Eingang_Stellung_1;
      AN    #in_Eingang_Stellung_2;
      O;
      A     DIX [AR2,P#0.5];	// Kennung "invers"
      AN    #in_Eingang_Stellung_1;
      AN    #in_Eingang_Stellung_2;
      );
      JC    disp;
// 14 = Störung, Stellung 2, nicht quittiert ==> rot/weiß
      L     14;
      A     #io_Stoerung;
      AN    #in_Quitt_Stoerung;
      A(;
      AN    DIX [AR2,P#0.5];	// Kennung "invers"
      AN    #in_Eingang_Stellung_1;	// (018) = Stellung 2 oder Keine
      O;
      A     DIX [AR2,P#0.5];	// Kennung "invers"
      AN    #in_Eingang_Stellung_2;	// (018) = Stellung 1 oder Keine
      );
      JC    disp;
// 15 = Störung, Stellung 1, nicht quittiert ==> rot/grün
      L     15;
      A     #io_Stoerung;
      AN    #in_Quitt_Stoerung;
      A(;
      AN    DIX [AR2,P#0.5];	// Kennung "invers"
      A     #in_Eingang_Stellung_1;
      O;
      A     DIX [AR2,P#0.5];	// Kennung "invers"
      A     #in_Eingang_Stellung_2;
      );
      JC    disp;
// 16 = Störung quittiert ==> rot
      L     16;
      A     #io_Stoerung;
      JC    disp;
NSV3: NOP   0;
NETWORK
TITLE = Objektstatus speichern (017)
//jm 20120907
      L     0;
disp: T     #Objektstatus;
NETWORK
TITLE = Daten in Struktur speichern
      A     #in_Anlage_ein;	// (021)
      =     DIX [AR2,P#4.5];	// (021) Anlage ein (Struktur)
      A     #in_Eingang_Stellung_1;
      =     DIX [AR2,P#2.2];	// Eingang Stellung 1 (Struktur)
      A     #in_Eingang_Stellung_2;
      =     DIX [AR2,P#2.3];	// Eingang Stellung 2 (Struktur)
      A     #io_Ausgang_Stellung_1;
      =     DIX [AR2,P#2.0];	// Ausgang Stellung 1 (Struktur)
      A     #io_Ausgang_Stellung_2;
      =     DIX [AR2,P#2.1];	// Ausgang Stellung 2 (Struktur)
      A     #io_Stellung_1_Betrieb;
      =     DIX [AR2,P#2.6];	// Stellung 1 in Betrieb (Struktur)
      A     #io_Stellung_2_Betrieb;
      =     DIX [AR2,P#2.7];	// Stellung 2 in Betrieb (Struktur)
      A     #io_Stoerung;
      =     DIX [AR2,P#3.0];	// Störung (Struktur)
      A     #Taktanzahl_erreicht;
      =     DIX [AR2,P#3.7];	// Taktanzahl erreicht (Struktur)
      A     #Taktausgang;
      =     DIX [AR2,P#4.3];	// Taktausgang (Struktur)
      L     #Zeitzaehler;
      T     DID [AR2,P#18.0];	// Impuls-/Pausezähler (Struktur)
      L     #Taktzaehler;
      T     DIW [AR2,P#24.0];	// Taktzähler (Struktur)
      L     #Objektstatus;	// (011)
      T     DIW [AR2,P#48.0];	// #Objektstatus  (Struktur)   // (011)
NETWORK
TITLE = ENDE
      NOP   0;
END_FUNCTION

